LIN {X 0,Y 324.27,Z 263.767,A -85,B 0,C 180,E1 -15871.54,E2 -15871.54} C_VEL
LIN {X 0,Y 321.442,Z 259.609,A -85,B 0,C 180,E1 -15872.86,E2 -15872.86} C_VEL
LIN {X 0,Y 318.492,Z 255.533,A -85,B 0,C 180,E1 -15874.441,E2 -15874.441} C_VEL
LIN {X 0,Y 315.534,Z 252.043,A -85,B 0,C 180,E1 -15876.317,E2 -15876.317} C_VEL
LIN {X 0,Y 314.496,Z 250.773,A -85,B 0,C 180,E1 -15877.111,E2 -15877.111} C_VEL
LIN {X 0,Y 311.264,Z 247.746,A -85,B 0,C 180,E1 -15880.434,E2 -15880.434} C_VEL
LIN {X 0,Y 310.658,Z 246.885,A -85,B 0,C 180,E1 -15881.705,E2 -15881.705} C_VEL
LIN {X 0,Y 310.882,Z 247.509,A -85,B 0,C 180,E1 -15884.492,E2 -15884.492} C_VEL
LIN {X 0,Y 311.343,Z 249.074,A -85,B 0,C 180,E1 -15887.373,E2 -15887.373} C_VEL
LIN {X 0,Y 311.812,Z 250.468,A -85,B 0,C 180,E1 -15888.852,E2 -15888.852} C_VEL
LIN {X 0,Y 315.445,Z 256.63,A -85,B 0,C 180,E1 -15892.27,E2 -15892.27} C_VEL
LIN {X 0,Y 317.186,Z 259.203,A -85,B 0,C 180,E1 -15893.415,E2 -15893.415} C_VEL
LIN {X 0,Y 321.138,Z 266.17,A -85,B 0,C 180,E1 -15895.657,E2 -15895.657} C_VEL
LIN {X 0,Y 324.404,Z 272.439,A -85,B 0,C 180,E1 -15897.229,E2 -15897.229} C_VEL
LIN {X 0,Y 327.131,Z 278.303,A -85,B 0,C 180,E1 -15898.426,E2 -15898.426} C_VEL
LIN {X 0,Y 329.213,Z 283.156,A -85,B 0,C 180,E1 -15899.287,E2 -15899.287} C_VEL
LIN {X 0,Y 330.879,Z 295.045,A -85,B 0,C 180,E1 -15900.451,E2 -15900.451} C_VEL
LIN {X 0,Y 331.883,Z 305.844,A -85,B 0,C 180,E1 -15901.326,E2 -15901.326} C_VEL
LIN {X 0,Y 331.943,Z 308.748,A -85,B 0,C 180,E1 -15901.513,E2 -15901.513} C_VEL
LIN {X 0,Y 325.93,Z 368.1,A -85,B 0,C 180,E1 -15903.808,E2 -15903.808} C_VEL
LIN {X 0,Y 323.729,Z 382.809,A -85,B 0,C 180,E1 -15904.61,E2 -15904.61} C_VEL
LIN {X 0,Y 321.291,Z 396.25,A -85,B 0,C 180,E1 -15905.613,E2 -15905.613} C_VEL
LIN {X 0,Y 318.7,Z 408.35,A -85,B 0,C 180,E1 -15906.784,E2 -15906.784} C_VEL
LIN {X 0,Y 316.184,Z 419.438,A -85,B 0,C 180,E1 -15908.14,E2 -15908.14} C_VEL
LIN {X 0,Y 313.663,Z 429.65,A -85,B 0,C 180,E1 -15909.677,E2 -15909.677} C_VEL
LIN {X 0,Y 311.064,Z 439.677,A -85,B 0,C 180,E1 -15911.559,E2 -15911.559} C_VEL
LIN {X 0,Y 308.863,Z 447.905,A -85,B 0,C 180,E1 -15913.474,E2 -15913.474} C_VEL
LIN {X 0,Y 307.172,Z 454.592,A -85,B 0,C 180,E1 -15915.422,E2 -15915.422} C_VEL
LIN {X 0,Y 305.752,Z 460.004,A -85,B 0,C 180,E1 -15917.385,E2 -15917.385} C_VEL
LIN {X 0,Y 304.767,Z 464.279,A -85,B 0,C 180,E1 -15919.368,E2 -15919.368} C_VEL
LIN {X 0,Y 304.309,Z 466.526,A -85,B 0,C 180,E1 -15920.695,E2 -15920.695} C_VEL
LIN {X 0,Y 303.954,Z 468.349,A -85,B 0,C 180,E1 -15922.024,E2 -15922.024} C_VEL
LIN {X 0,Y 303.66,Z 470.501,A -85,B 0,C 180,E1 -15924.387,E2 -15924.387} C_VEL
LIN {X 0,Y 303.654,Z 471.167,A -85,B 0,C 180,E1 -15926.017,E2 -15926.017} C_VEL
LIN {X 0,Y 303.655,Z 471.261,A -85,B 0,C 180,E1 -15927.345,E2 -15927.345} C_VEL
LIN {X 0,Y 303.985,Z 470.229,A -85,B 0,C 180,E1 -15929.999,E2 -15929.999} C_VEL
LIN {X 0,Y 303.726,Z 470.328,A -85,B 0,C 180,E1 -15932.651,E2 -15932.651} C_VEL
LIN {X 0,Y 303.689,Z 469.744,A -85,B 0,C 180,E1 -15933.98,E2 -15933.98} C_VEL
LIN {X 0,Y 303.728,Z 468.388,A -85,B 0,C 180,E1 -15935.742,E2 -15935.742} C_VEL
LIN {X 0,Y 303.923,Z 465.595,A -85,B 0,C 180,E1 -15937.974,E2 -15937.974} C_VEL
LIN {X 0,Y 304.374,Z 462.049,A -85,B 0,C 180,E1 -15939.971,E2 -15939.971} C_VEL
LIN {X 0,Y 305.1,Z 457.403,A -85,B 0,C 180,E1 -15941.964,E2 -15941.964} C_VEL
LIN {X 0,Y 306.576,Z 450.407,A -85,B 0,C 180,E1 -15944.265,E2 -15944.265} C_VEL
LIN {X 0,Y 308.034,Z 442.766,A -85,B 0,C 180,E1 -15946.251,E2 -15946.251} C_VEL
LIN {X 0,Y 309.524,Z 435.145,A -85,B 0,C 180,E1 -15947.849,E2 -15947.849} C_VEL
LIN {X 0,Y 311.634,Z 424.665,A -85,B 0,C 180,E1 -15949.599,E2 -15949.599} C_VEL
LIN {X 0,Y 313.577,Z 414.013,A -85,B 0,C 180,E1 -15951.012,E2 -15951.012} C_VEL
LIN {X 0,Y 315.419,Z 401.913,A -85,B 0,C 180,E1 -15952.257,E2 -15952.257} C_VEL
LIN {X 0,Y 317.041,Z 390.09,A -85,B 0,C 180,E1 -15953.169,E2 -15953.169} C_VEL
LIN {X 0,Y 318.385,Z 378.012,A -85,B 0,C 180,E1 -15953.841,E2 -15953.841} C_VEL
LIN {X 0,Y 319.265,Z 364.396,A -85,B 0,C 180,E1 -15954.332,E2 -15954.332} C_VEL
LIN {X 0,Y 320.858,Z 303.853,A -85,B 0,C 180,E1 -15955.738,E2 -15955.738} C_VEL
LIN {X 0,Y 317.941,Z 282.581,A -85,B 0,C 180,E1 -15956.599,E2 -15956.599} C_VEL
LIN {X 0,Y 313.357,Z 256.247,A -85,B 0,C 180,E1 -15957.81,E2 -15957.81} C_VEL
LIN {X 0,Y 310.41,Z 248.436,A -85,B 0,C 180,E1 -15958.367,E2 -15958.367} C_VEL
LIN {X 0,Y 306.974,Z 238.832,A -85,B 0,C 180,E1 -15959.129,E2 -15959.129} C_VEL
LIN {X 0,Y 305.494,Z 231.423,A -85,B 0,C 180,E1 -15961.306,E2 -15961.306} C_VEL
LIN {X 0,Y 305.457,Z 231.411,A -85,B 0,C 180,E1 -15965.112,E2 -15965.112} C_VEL
LIN {X 0,Y 305.405,Z 231.432,A -85,B 0,C 180,E1 -15968.518,E2 -15968.518} C_VEL
LIN {X 0,Y 305.429,Z 231.43,A -85,B 0,C 180,E1 -15972.581,E2 -15972.581} C_VEL
LIN {X 0,Y 305.415,Z 231.439,A -85,B 0,C 180,E1 -15976.343,E2 -15976.343} C_VEL
LIN {X 0,Y 305.402,Z 231.436,A -85,B 0,C 180,E1 -15979.884,E2 -15979.884} C_VEL
LIN {X 0,Y 305.455,Z 231.413,A -85,B 0,C 180,E1 -15983.635,E2 -15983.635} C_VEL
LIN {X 0,Y 305.457,Z 231.429,A -85,B 0,C 180,E1 -15986.482,E2 -15986.482} C_VEL
LIN {X 0,Y 305.409,Z 231.42,A -85,B 0,C 180,E1 -15989.585,E2 -15989.585} C_VEL
LIN {X 0,Y 305.438,Z 231.423,A -85,B 0,C 180,E1 -15992.601,E2 -15992.601} C_VEL
LIN {X 0,Y 305.464,Z 231.423,A -85,B 0,C 180,E1 -15995.535,E2 -15995.535} C_VEL
LIN {X 0,Y 305.454,Z 231.402,A -85,B 0,C 180,E1 -15998.4,E2 -15998.4} C_VEL
LIN {X 0,Y 305.526,Z 231.425,A -85,B 0,C 180,E1 -16002.6,E2 -16002.6} C_VEL
LIN {X 0,Y 305.617,Z 231.385,A -85,B 0,C 180,E1 -16005.348,E2 -16005.348} C_VEL
LIN {X 0,Y 305.615,Z 231.414,A -85,B 0,C 180,E1 -16009.399,E2 -16009.399} C_VEL
LIN {X 0,Y 305.736,Z 231.392,A -85,B 0,C 180,E1 -16012.073,E2 -16012.073} C_VEL
LIN {X 0,Y 305.651,Z 231.378,A -85,B 0,C 180,E1 -16014.723,E2 -16014.723} C_VEL
LIN {X 0,Y 305.929,Z 231.374,A -85,B 0,C 180,E1 -16018.684,E2 -16018.684} C_VEL
LIN {X 0,Y 305.94,Z 231.353,A -85,B 0,C 180,E1 -16021.317,E2 -16021.317} C_VEL
LIN {X 0,Y 305.833,Z 231.384,A -85,B 0,C 180,E1 -16026.598,E2 -16026.598} C_VEL
LIN {X 0,Y 305.696,Z 231.382,A -85,B 0,C 180,E1 -16029.261,E2 -16029.261} C_VEL
LIN {X 0,Y 305.579,Z 231.414,A -85,B 0,C 180,E1 -16033.297,E2 -16033.297} C_VEL
LIN {X 0,Y 305.544,Z 231.409,A -85,B 0,C 180,E1 -16036.023,E2 -16036.023} C_VEL
LIN {X 0,Y 305.54,Z 231.417,A -85,B 0,C 180,E1 -16039.43,E2 -16039.43} C_VEL
LIN {X 0,Y 305.484,Z 231.417,A -85,B 0,C 180,E1 -16043.042,E2 -16043.042} C_VEL
LIN {X 0,Y 305.54,Z 231.425,A -85,B 0,C 180,E1 -16046.228,E2 -16046.228} C_VEL
LIN {X 0,Y 305.481,Z 231.419,A -85,B 0,C 180,E1 -16049.048,E2 -16049.048} C_VEL
LIN {X 0,Y 305.436,Z 231.44,A -85,B 0,C 180,E1 -16051.954,E2 -16051.954} C_VEL
LIN {X 0,Y 305.457,Z 231.43,A -85,B 0,C 180,E1 -16055.114,E2 -16055.114} C_VEL
LIN {X 0,Y 305.445,Z 231.43,A -85,B 0,C 180,E1 -16058.53,E2 -16058.53} C_VEL
LIN {X 0,Y 305.452,Z 231.432,A -85,B 0,C 180,E1 -16062.588,E2 -16062.588} C_VEL
LIN {X 0,Y 305.409,Z 231.439,A -85,B 0,C 180,E1 -16066.937,E2 -16066.937} C_VEL
LIN {X 0,Y 306.456,Z 234.33,A -85,B 0,C 180,E1 -16067.175,E2 -16067.175} C_VEL
LIN {X 0,Y 308.07,Z 236.957,A -85,B 0,C 180,E1 -16067.448,E2 -16067.448} C_VEL
LIN {X 0,Y 316.648,Z 252.215,A -85,B 0,C 180,E1 -16068.873,E2 -16068.873} C_VEL
LIN {X 0,Y 322.599,Z 264.535,A -85,B 0,C 180,E1 -16069.845,E2 -16069.845} C_VEL
LIN {X 0,Y 320.216,Z 341.058,A -85,B 0,C 180,E1 -16071.589,E2 -16071.589} C_VEL
LIN {X 0,Y 319.435,Z 354.384,A -85,B 0,C 180,E1 -16072.142,E2 -16072.142} C_VEL
LIN {X 0,Y 318.476,Z 365.661,A -85,B 0,C 180,E1 -16072.842,E2 -16072.842} C_VEL
LIN {X 0,Y 317.019,Z 377.635,A -85,B 0,C 180,E1 -16073.827,E2 -16073.827} C_VEL
LIN {X 0,Y 315.458,Z 388.546,A -85,B 0,C 180,E1 -16074.994,E2 -16074.994} C_VEL
LIN {X 0,Y 313.687,Z 398.497,A -85,B 0,C 180,E1 -16076.325,E2 -16076.325} C_VEL
LIN {X 0,Y 311.761,Z 408.517,A -85,B 0,C 180,E1 -16078.013,E2 -16078.013} C_VEL
LIN {X 0,Y 310.025,Z 416.996,A -85,B 0,C 180,E1 -16079.795,E2 -16079.795} C_VEL
LIN {X 0,Y 308.34,Z 424.504,A -85,B 0,C 180,E1 -16081.776,E2 -16081.776} C_VEL
LIN {X 0,Y 307.033,Z 430.143,A -85,B 0,C 180,E1 -16083.635,E2 -16083.635} C_VEL
LIN {X 0,Y 305.974,Z 434.812,A -85,B 0,C 180,E1 -16085.58,E2 -16085.58} C_VEL
LIN {X 0,Y 305.06,Z 438.66,A -85,B 0,C 180,E1 -16087.692,E2 -16087.692} C_VEL
LIN {X 0,Y 304.37,Z 441.306,A -85,B 0,C 180,E1 -16089.737,E2 -16089.737} C_VEL
LIN {X 0,Y 303.992,Z 442.756,A -85,B 0,C 180,E1 -16091.422,E2 -16091.422} C_VEL
LIN {X 0,Y 303.63,Z 443.679,A -85,B 0,C 180,E1 -16093.875,E2 -16093.875} C_VEL
LIN {X 0,Y 303.576,Z 443.218,A -85,B 0,C 180,E1 -16096.493,E2 -16096.493} C_VEL
LIN {X 0,Y 303.6,Z 442.239,A -85,B 0,C 180,E1 -16097.976,E2 -16097.976} C_VEL
LIN {X 0,Y 303.652,Z 440.927,A -85,B 0,C 180,E1 -16099.331,E2 -16099.331} C_VEL
LIN {X 0,Y 303.933,Z 438.132,A -85,B 0,C 180,E1 -16101.357,E2 -16101.357} C_VEL
LIN {X 0,Y 304.331,Z 434.302,A -85,B 0,C 180,E1 -16103.371,E2 -16103.371} C_VEL
LIN {X 0,Y 304.804,Z 429.35,A -85,B 0,C 180,E1 -16105.373,E2 -16105.373} C_VEL
LIN {X 0,Y 305.504,Z 423.101,A -85,B 0,C 180,E1 -16107.364,E2 -16107.364} C_VEL
LIN {X 0,Y 306.468,Z 415.263,A -85,B 0,C 180,E1 -16109.344,E2 -16109.344} C_VEL
LIN {X 0,Y 307.432,Z 407.282,A -85,B 0,C 180,E1 -16110.984,E2 -16110.984} C_VEL
LIN {X 0,Y 308.623,Z 397.563,A -85,B 0,C 180,E1 -16112.612,E2 -16112.612} C_VEL
LIN {X 0,Y 309.875,Z 386.849,A -85,B 0,C 180,E1 -16114.037,E2 -16114.037} C_VEL
LIN {X 0,Y 310.915,Z 375.975,A -85,B 0,C 180,E1 -16115.189,E2 -16115.189} C_VEL
LIN {X 0,Y 311.705,Z 364.413,A -85,B 0,C 180,E1 -16116.149,E2 -16116.149} C_VEL
LIN {X 0,Y 312.482,Z 351.83,A -85,B 0,C 180,E1 -16116.904,E2 -16116.904} C_VEL
LIN {X 0,Y 312.982,Z 338.785,A -85,B 0,C 180,E1 -16117.42,E2 -16117.42} C_VEL
LIN {X 0,Y 314.728,Z 259.21,A -85,B 0,C 180,E1 -16119.23,E2 -16119.23} C_VEL
LIN {X 0,Y 313.342,Z 251.333,A -85,B 0,C 180,E1 -16119.507,E2 -16119.507} C_VEL
LIN {X 0,Y 306.45,Z 233.925,A -85,B 0,C 180,E1 -16120.389,E2 -16120.389} C_VEL
LIN {X 0,Y 305.654,Z 231.414,A -85,B 0,C 180,E1 -16120.548,E2 -16120.548} C_VEL
LIN {X 0,Y 305.644,Z 231.411,A -85,B 0,C 180,E1 -16125.036,E2 -16125.036} C_VEL
LIN {X 0,Y 305.586,Z 231.419,A -85,B 0,C 180,E1 -16128.784,E2 -16128.784} C_VEL
LIN {X 0,Y 305.477,Z 231.43,A -85,B 0,C 180,E1 -16133.033,E2 -16133.033} C_VEL
LIN {X 0,Y 305.458,Z 231.436,A -85,B 0,C 180,E1 -16136.191,E2 -16136.191} C_VEL
LIN {X 0,Y 305.431,Z 231.437,A -85,B 0,C 180,E1 -16139.027,E2 -16139.027} C_VEL
LIN {X 0,Y 305.443,Z 231.439,A -85,B 0,C 180,E1 -16141.954,E2 -16141.954} C_VEL
LIN {X 0,Y 305.467,Z 231.432,A -85,B 0,C 180,E1 -16145.114,E2 -16145.114} C_VEL
LIN {X 0,Y 305.439,Z 231.436,A -85,B 0,C 180,E1 -16148.525,E2 -16148.525} C_VEL
LIN {X 0,Y 305.44,Z 231.432,A -85,B 0,C 180,E1 -16152.582,E2 -16152.582} C_VEL
LIN {X 0,Y 305.426,Z 231.437,A -85,B 0,C 180,E1 -16156.344,E2 -16156.344} C_VEL
LIN {X 0,Y 305.4,Z 231.439,A -85,B 0,C 180,E1 -16159.037,E2 -16159.037} C_VEL
LIN {X 0,Y 304.753,Z 231.522,A -85,B 0,C 180,E1 -16160.138,E2 -16160.138} C_VEL
LIN {X 0,Y 301.902,Z 231.875,A -85,B 0,C 180,E1 -16161.931,E2 -16161.931} C_VEL
LIN {X 0,Y 299.485,Z 232.178,A -85,B 0,C 180,E1 -16163.386,E2 -16163.386} C_VEL
LIN {X 0,Y 298.469,Z 232.303,A -85,B 0,C 180,E1 -16164.513,E2 -16164.513} C_VEL
LIN {X 0,Y 298.398,Z 232.309,A -85,B 0,C 180,E1 -16164.894,E2 -16164.894} C_VEL
LIN {X 0,Y 298.377,Z 232.317,A -85,B 0,C 180,E1 -16168.789,E2 -16168.789} C_VEL
LIN {X 0,Y 298.41,Z 232.302,A -85,B 0,C 180,E1 -16171.898,E2 -16171.898} C_VEL
LIN {X 0,Y 298.471,Z 232.351,A -85,B 0,C 180,E1 -16175.457,E2 -16175.457} C_VEL
LIN {X 0,Y 298.728,Z 233.608,A -85,B 0,C 180,E1 -16175.791,E2 -16175.791} C_VEL
LIN {X 0,Y 304.574,Z 256.081,A -85,B 0,C 180,E1 -16176.845,E2 -16176.845} C_VEL
LIN {X 0,Y 305.328,Z 261.998,A -85,B 0,C 180,E1 -16177.086,E2 -16177.086} C_VEL
LIN {X 0,Y 302.456,Z 342.479,A -85,B 0,C 180,E1 -16179.911,E2 -16179.911} C_VEL
LIN {X 0,Y 301.986,Z 355.703,A -85,B 0,C 180,E1 -16180.632,E2 -16180.632} C_VEL
LIN {X 0,Y 301.269,Z 369.111,A -85,B 0,C 180,E1 -16181.643,E2 -16181.643} C_VEL
LIN {X 0,Y 300.468,Z 381.148,A -85,B 0,C 180,E1 -16182.824,E2 -16182.824} C_VEL
LIN {X 0,Y 299.696,Z 391.71,A -85,B 0,C 180,E1 -16184.116,E2 -16184.116} C_VEL
LIN {X 0,Y 298.948,Z 402.266,A -85,B 0,C 180,E1 -16185.709,E2 -16185.709} C_VEL
LIN {X 0,Y 298.245,Z 411.532,A -85,B 0,C 180,E1 -16187.41,E2 -16187.41} C_VEL
LIN {X 0,Y 297.714,Z 419.213,A -85,B 0,C 180,E1 -16189.114,E2 -16189.114} C_VEL
LIN {X 0,Y 297.237,Z 426.724,A -85,B 0,C 180,E1 -16191.159,E2 -16191.159} C_VEL
LIN {X 0,Y 296.932,Z 432.717,A -85,B 0,C 180,E1 -16193.203,E2 -16193.203} C_VEL
LIN {X 0,Y 296.744,Z 437.411,A -85,B 0,C 180,E1 -16195.245,E2 -16195.245} C_VEL
LIN {X 0,Y 296.681,Z 440.952,A -85,B 0,C 180,E1 -16197.284,E2 -16197.284} C_VEL
LIN {X 0,Y 296.631,Z 442.74,A -85,B 0,C 180,E1 -16198.642,E2 -16198.642} C_VEL
LIN {X 0,Y 296.695,Z 444.045,A -85,B 0,C 180,E1 -16200,E2 -16200} C_VEL
LIN {X 0,Y 296.858,Z 444.911,A -85,B 0,C 180,E1 -16201.356,E2 -16201.356} C_VEL
LIN {X 0,Y 297.102,Z 445.37,A -85,B 0,C 180,E1 -16202.711,E2 -16202.711} C_VEL
LIN {X 0,Y 297.47,Z 445.402,A -85,B 0,C 180,E1 -16204.064,E2 -16204.064} C_VEL
LIN {X 0,Y 297.933,Z 444.971,A -85,B 0,C 180,E1 -16205.414,E2 -16205.414} C_VEL
LIN {X 0,Y 298.231,Z 444.155,A -85,B 0,C 180,E1 -16206.767,E2 -16206.767} C_VEL
LIN {X 0,Y 298.552,Z 442.95,A -85,B 0,C 180,E1 -16208.119,E2 -16208.119} C_VEL
LIN {X 0,Y 300.197,Z 439.612,A -85,B 0,C 180,E1 -16210.487,E2 -16210.487} C_VEL
LIN {X 0,Y 301.927,Z 434.969,A -85,B 0,C 180,E1 -16212.775,E2 -16212.775} C_VEL
LIN {X 0,Y 304.13,Z 428.717,A -85,B 0,C 180,E1 -16215.068,E2 -16215.068} C_VEL
LIN {X 0,Y 306.32,Z 421.893,A -85,B 0,C 180,E1 -16217.009,E2 -16217.009} C_VEL
LIN {X 0,Y 308.873,Z 413.464,A -85,B 0,C 180,E1 -16218.919,E2 -16218.919} C_VEL
LIN {X 0,Y 311.286,Z 404.929,A -85,B 0,C 180,E1 -16220.484,E2 -16220.484} C_VEL
LIN {X 0,Y 313.958,Z 394.59,A -85,B 0,C 180,E1 -16222.021,E2 -16222.021} C_VEL
LIN {X 0,Y 316.768,Z 381.851,A -85,B 0,C 180,E1 -16223.538,E2 -16223.538} C_VEL
LIN {X 0,Y 319.27,Z 368.719,A -85,B 0,C 180,E1 -16224.723,E2 -16224.723} C_VEL
LIN {X 0,Y 321.125,Z 356.231,A -85,B 0,C 180,E1 -16225.61,E2 -16225.61} C_VEL
LIN {X 0,Y 322.948,Z 340.967,A -85,B 0,C 180,E1 -16226.364,E2 -16226.364} C_VEL
LIN {X 0,Y 329.392,Z 284.527,A -85,B 0,C 180,E1 -16228.59,E2 -16228.59} C_VEL
LIN {X 0,Y 325.775,Z 277.054,A -85,B 0,C 180,E1 -16230.035,E2 -16230.035} C_VEL
LIN {X 0,Y 321.791,Z 270.367,A -85,B 0,C 180,E1 -16231.752,E2 -16231.752} C_VEL
LIN {X 0,Y 318.626,Z 265.727,A -85,B 0,C 180,E1 -16233.288,E2 -16233.288} C_VEL
LIN {X 0,Y 315.758,Z 261.708,A -85,B 0,C 180,E1 -16234.924,E2 -16234.924} C_VEL
LIN {X 0,Y 313.045,Z 258.146,A -85,B 0,C 180,E1 -16236.827,E2 -16236.827} C_VEL
LIN {X 0,Y 311.199,Z 256.452,A -85,B 0,C 180,E1 -16238.376,E2 -16238.376} C_VEL
LIN {X 0,Y 309.035,Z 253.983,A -85,B 0,C 180,E1 -16241.366,E2 -16241.366} C_VEL
LIN {X 0,Y 308.261,Z 254.006,A -85,B 0,C 180,E1 -16244.08,E2 -16244.08} C_VEL
LIN {X 0,Y 308.771,Z 255.362,A -85,B 0,C 180,E1 -16246.749,E2 -16246.749} C_VEL
LIN {X 0,Y 309.859,Z 257.192,A -85,B 0,C 180,E1 -16248.618,E2 -16248.618} C_VEL
LIN {X 0,Y 313.257,Z 263.264,A -85,B 0,C 180,E1 -16252.027,E2 -16252.027} C_VEL
LIN {X 0,Y 314.664,Z 265.534,A -85,B 0,C 180,E1 -16253.024,E2 -16253.024} C_VEL
LIN {X 0,Y 318.17,Z 272.075,A -85,B 0,C 180,E1 -16255.176,E2 -16255.176} C_VEL
LIN {X 0,Y 321.172,Z 278.16,A -85,B 0,C 180,E1 -16256.732,E2 -16256.732} C_VEL
LIN {X 0,Y 323.667,Z 283.829,A -85,B 0,C 180,E1 -16257.919,E2 -16257.919} C_VEL
LIN {X 0,Y 325.18,Z 287.739,A -85,B 0,C 180,E1 -16258.614,E2 -16258.614} C_VEL
LIN {X 0,Y 326.58,Z 299.644,A -85,B 0,C 180,E1 -16259.794,E2 -16259.794} C_VEL
LIN {X 0,Y 327.257,Z 309.221,A -85,B 0,C 180,E1 -16260.574,E2 -16260.574} C_VEL
LIN {X 0,Y 320.93,Z 367.302,A -85,B 0,C 180,E1 -16262.884,E2 -16262.884} C_VEL
LIN {X 0,Y 318.79,Z 381.297,A -85,B 0,C 180,E1 -16263.66,E2 -16263.66} C_VEL
LIN {X 0,Y 316.461,Z 393.138,A -85,B 0,C 180,E1 -16264.513,E2 -16264.513} C_VEL
LIN {X 0,Y 313.705,Z 405.712,A -85,B 0,C 180,E1 -16265.689,E2 -16265.689} C_VEL
LIN {X 0,Y 310.879,Z 417.125,A -85,B 0,C 180,E1 -16267.046,E2 -16267.046} C_VEL
LIN {X 0,Y 308.187,Z 427.579,A -85,B 0,C 180,E1 -16268.599,E2 -16268.599} C_VEL
LIN {X 0,Y 305.749,Z 436.315,A -85,B 0,C 180,E1 -16270.18,E2 -16270.18} C_VEL
LIN {X 0,Y 303.163,Z 445.032,A -85,B 0,C 180,E1 -16272.113,E2 -16272.113} C_VEL
LIN {X 0,Y 301.249,Z 452.123,A -85,B 0,C 180,E1 -16274.089,E2 -16274.089} C_VEL
LIN {X 0,Y 299.216,Z 458.804,A -85,B 0,C 180,E1 -16276.414,E2 -16276.414} C_VEL
LIN {X 0,Y 298.098,Z 463.24,A -85,B 0,C 180,E1 -16278.438,E2 -16278.438} C_VEL
LIN {X 0,Y 297.281,Z 466.614,A -85,B 0,C 180,E1 -16280.473,E2 -16280.473} C_VEL
LIN {X 0,Y 296.895,Z 468.311,A -85,B 0,C 180,E1 -16281.833,E2 -16281.833} C_VEL
LIN {X 0,Y 296.588,Z 470.328,A -85,B 0,C 180,E1 -16284.406,E2 -16284.406} C_VEL
LIN {X 0,Y 296.568,Z 470.839,A -85,B 0,C 180,E1 -16285.922,E2 -16285.922} C_VEL
LIN {X 0,Y 296.578,Z 470.815,A -85,B 0,C 180,E1 -16287.282,E2 -16287.282} C_VEL
LIN {X 0,Y 296.889,Z 469.87,A -85,B 0,C 180,E1 -16289.999,E2 -16289.999} C_VEL
LIN {X 0,Y 296.644,Z 470.033,A -85,B 0,C 180,E1 -16292.714,E2 -16292.714} C_VEL
LIN {X 0,Y 296.603,Z 469.487,A -85,B 0,C 180,E1 -16294.075,E2 -16294.075} C_VEL
LIN {X 0,Y 296.622,Z 468.346,A -85,B 0,C 180,E1 -16295.659,E2 -16295.659} C_VEL
LIN {X 0,Y 296.862,Z 465.434,A -85,B 0,C 180,E1 -16298.165,E2 -16298.165} C_VEL
LIN {X 0,Y 297.361,Z 461.943,A -85,B 0,C 180,E1 -16300.209,E2 -16300.209} C_VEL
LIN {X 0,Y 298.121,Z 457.363,A -85,B 0,C 180,E1 -16302.248,E2 -16302.248} C_VEL
LIN {X 0,Y 299.691,Z 450.436,A -85,B 0,C 180,E1 -16304.6,E2 -16304.6} C_VEL
LIN {X 0,Y 301.158,Z 443.106,A -85,B 0,C 180,E1 -16306.573,E2 -16306.573} C_VEL
LIN {X 0,Y 302.781,Z 435.35,A -85,B 0,C 180,E1 -16308.26,E2 -16308.26} C_VEL
LIN {X 0,Y 304.754,Z 426.07,A -85,B 0,C 180,E1 -16309.885,E2 -16309.885} C_VEL
LIN {X 0,Y 306.792,Z 415.77,A -85,B 0,C 180,E1 -16311.324,E2 -16311.324} C_VEL
LIN {X 0,Y 308.654,Z 404.364,A -85,B 0,C 180,E1 -16312.595,E2 -16312.595} C_VEL
LIN {X 0,Y 310.435,Z 392.286,A -85,B 0,C 180,E1 -16313.603,E2 -16313.603} C_VEL
LIN {X 0,Y 312.032,Z 378.901,A -85,B 0,C 180,E1 -16314.402,E2 -16314.402} C_VEL
LIN {X 0,Y 312.967,Z 366.327,A -85,B 0,C 180,E1 -16314.899,E2 -16314.899} C_VEL
LIN {X 0,Y 314.722,Z 304.889,A -85,B 0,C 180,E1 -16316.36,E2 -16316.36} C_VEL
LIN {X 0,Y 312.132,Z 285.348,A -85,B 0,C 180,E1 -16317.168,E2 -16317.168} C_VEL
LIN {X 0,Y 307.592,Z 258.654,A -85,B 0,C 180,E1 -16318.424,E2 -16318.424} C_VEL
LIN {X 0,Y 301.295,Z 242.01,A -85,B 0,C 180,E1 -16319.725,E2 -16319.725} C_VEL
LIN {X 0,Y 299.357,Z 236.961,A -85,B 0,C 180,E1 -16320.186,E2 -16320.186} C_VEL
LIN {X 0,Y 299.192,Z 236.151,A -85,B 0,C 180,E1 -16320.29,E2 -16320.29} C_VEL
LIN {X 0,Y 298.455,Z 232.294,A -85,B 0,C 180,E1 -16321.49,E2 -16321.49} C_VEL
LIN {X 0,Y 298.423,Z 232.277,A -85,B 0,C 180,E1 -16324.486,E2 -16324.486} C_VEL
LIN {X 0,Y 298.386,Z 232.313,A -85,B 0,C 180,E1 -16327.76,E2 -16327.76} C_VEL
LIN {X 0,Y 298.342,Z 232.324,A -85,B 0,C 180,E1 -16331.266,E2 -16331.266} C_VEL
LIN {X 0,Y 298.348,Z 232.319,A -85,B 0,C 180,E1 -16335.034,E2 -16335.034} C_VEL
LIN {X 0,Y 298.34,Z 232.305,A -85,B 0,C 180,E1 -16338.92,E2 -16338.92} C_VEL
LIN {X 0,Y 298.391,Z 232.31,A -85,B 0,C 180,E1 -16342.238,E2 -16342.238} C_VEL
LIN {X 0,Y 298.4,Z 232.299,A -85,B 0,C 180,E1 -16345.58,E2 -16345.58} C_VEL
LIN {X 0,Y 298.364,Z 232.305,A -85,B 0,C 180,E1 -16348.788,E2 -16348.788} C_VEL
LIN {X 0,Y 298.39,Z 232.293,A -85,B 0,C 180,E1 -16351.897,E2 -16351.897} C_VEL
LIN {X 0,Y 298.429,Z 232.305,A -85,B 0,C 180,E1 -16354.919,E2 -16354.919} C_VEL
LIN {X 0,Y 298.391,Z 232.28,A -85,B 0,C 180,E1 -16357.862,E2 -16357.862} C_VEL
LIN {X 0,Y 298.455,Z 232.299,A -85,B 0,C 180,E1 -16360.751,E2 -16360.751} C_VEL
LIN {X 0,Y 298.577,Z 232.265,A -85,B 0,C 180,E1 -16364.994,E2 -16364.994} C_VEL
LIN {X 0,Y 298.574,Z 232.291,A -85,B 0,C 180,E1 -16369.146,E2 -16369.146} C_VEL
LIN {X 0,Y 298.688,Z 232.273,A -85,B 0,C 180,E1 -16371.884,E2 -16371.884} C_VEL
LIN {X 0,Y 298.621,Z 232.253,A -85,B 0,C 180,E1 -16374.598,E2 -16374.598} C_VEL
LIN {X 0,Y 298.897,Z 232.25,A -85,B 0,C 180,E1 -16378.653,E2 -16378.653} C_VEL
LIN {X 0,Y 298.906,Z 232.228,A -85,B 0,C 180,E1 -16381.348,E2 -16381.348} C_VEL
LIN {X 0,Y 298.778,Z 232.262,A -85,B 0,C 180,E1 -16386.755,E2 -16386.755} C_VEL
LIN {X 0,Y 298.627,Z 232.259,A -85,B 0,C 180,E1 -16389.483,E2 -16389.483} C_VEL
LIN {X 0,Y 298.538,Z 232.293,A -85,B 0,C 180,E1 -16393.616,E2 -16393.616} C_VEL
LIN {X 0,Y 298.479,Z 232.285,A -85,B 0,C 180,E1 -16396.413,E2 -16396.413} C_VEL
LIN {X 0,Y 298.481,Z 232.298,A -85,B 0,C 180,E1 -16399.643,E2 -16399.643} C_VEL
LIN {X 0,Y 298.451,Z 232.289,A -85,B 0,C 180,E1 -16403.599,E2 -16403.599} C_VEL
LIN {X 0,Y 298.483,Z 232.304,A -85,B 0,C 180,E1 -16406.576,E2 -16406.576} C_VEL
LIN {X 0,Y 298.41,Z 232.299,A -85,B 0,C 180,E1 -16409.643,E2 -16409.643} C_VEL
LIN {X 0,Y 298.389,Z 232.314,A -85,B 0,C 180,E1 -16412.802,E2 -16412.802} C_VEL
LIN {X 0,Y 298.442,Z 232.314,A -85,B 0,C 180,E1 -16416.809,E2 -16416.809} C_VEL
LIN {X 0,Y 298.382,Z 232.315,A -85,B 0,C 180,E1 -16421.089,E2 -16421.089} C_VEL
LIN {X 0,Y 298.394,Z 232.316,A -85,B 0,C 180,E1 -16423.105,E2 -16423.105} C_VEL
LIN {X 0,Y 298.36,Z 232.321,A -85,B 0,C 180,E1 -16426.047,E2 -16426.047} C_VEL
LIN {X 0,Y 299.336,Z 235.105,A -85,B 0,C 180,E1 -16426.278,E2 -16426.278} C_VEL
LIN {X 0,Y 301.106,Z 237.894,A -85,B 0,C 180,E1 -16426.593,E2 -16426.593} C_VEL
LIN {X 0,Y 310.001,Z 253.515,A -85,B 0,C 180,E1 -16428.137,E2 -16428.137} C_VEL
LIN {X 0,Y 316.428,Z 266.345,A -85,B 0,C 180,E1 -16429.222,E2 -16429.222} C_VEL
LIN {X 0,Y 314.031,Z 341.028,A -85,B 0,C 180,E1 -16430.956,E2 -16430.956} C_VEL
LIN {X 0,Y 313.272,Z 353.948,A -85,B 0,C 180,E1 -16431.49,E2 -16431.49} C_VEL
LIN {X 0,Y 312.243,Z 365.654,A -85,B 0,C 180,E1 -16432.216,E2 -16432.216} C_VEL
LIN {X 0,Y 310.778,Z 377.333,A -85,B 0,C 180,E1 -16433.184,E2 -16433.184} C_VEL
LIN {X 0,Y 309.151,Z 388.375,A -85,B 0,C 180,E1 -16434.373,E2 -16434.373} C_VEL
LIN {X 0,Y 307.297,Z 398.436,A -85,B 0,C 180,E1 -16435.726,E2 -16435.726} C_VEL
LIN {X 0,Y 305.422,Z 407.608,A -85,B 0,C 180,E1 -16437.267,E2 -16437.267} C_VEL
LIN {X 0,Y 303.614,Z 416.138,A -85,B 0,C 180,E1 -16439.048,E2 -16439.048} C_VEL
LIN {X 0,Y 301.772,Z 424.05,A -85,B 0,C 180,E1 -16441.104,E2 -16441.104} C_VEL
LIN {X 0,Y 300.283,Z 430.177,A -85,B 0,C 180,E1 -16443.132,E2 -16443.132} C_VEL
LIN {X 0,Y 299.204,Z 434.646,A -85,B 0,C 180,E1 -16444.99,E2 -16444.99} C_VEL
LIN {X 0,Y 298.395,Z 437.922,A -85,B 0,C 180,E1 -16446.717,E2 -16446.717} C_VEL
LIN {X 0,Y 297.424,Z 441.378,A -85,B 0,C 180,E1 -16449.242,E2 -16449.242} C_VEL
LIN {X 0,Y 296.943,Z 443.077,A -85,B 0,C 180,E1 -16451.213,E2 -16451.213} C_VEL
LIN {X 0,Y 296.578,Z 443.973,A -85,B 0,C 180,E1 -16453.481,E2 -16453.481} C_VEL
LIN {X 0,Y 296.465,Z 443.974,A -85,B 0,C 180,E1 -16454.886,E2 -16454.886} C_VEL
LIN {X 0,Y 296.478,Z 443.54,A -85,B 0,C 180,E1 -16456.389,E2 -16456.389} C_VEL
LIN {X 0,Y 296.493,Z 442.75,A -85,B 0,C 180,E1 -16457.684,E2 -16457.684} C_VEL
LIN {X 0,Y 296.537,Z 441.492,A -85,B 0,C 180,E1 -16459.072,E2 -16459.072} C_VEL
LIN {X 0,Y 296.799,Z 438.81,A -85,B 0,C 180,E1 -16461.148,E2 -16461.148} C_VEL
LIN {X 0,Y 297.213,Z 434.928,A -85,B 0,C 180,E1 -16463.294,E2 -16463.294} C_VEL
LIN {X 0,Y 297.672,Z 430.271,A -85,B 0,C 180,E1 -16465.262,E2 -16465.262} C_VEL
LIN {X 0,Y 298.382,Z 424.179,A -85,B 0,C 180,E1 -16467.301,E2 -16467.301} C_VEL
LIN {X 0,Y 299.348,Z 416.56,A -85,B 0,C 180,E1 -16469.329,E2 -16469.329} C_VEL
LIN {X 0,Y 300.543,Z 407.023,A -85,B 0,C 180,E1 -16471.341,E2 -16471.341} C_VEL
LIN {X 0,Y 301.81,Z 397.14,A -85,B 0,C 180,E1 -16473.005,E2 -16473.005} C_VEL
LIN {X 0,Y 303.157,Z 385.626,A -85,B 0,C 180,E1 -16474.535,E2 -16474.535} C_VEL
LIN {X 0,Y 304.165,Z 375.162,A -85,B 0,C 180,E1 -16475.637,E2 -16475.637} C_VEL
LIN {X 0,Y 305.006,Z 363.172,A -85,B 0,C 180,E1 -16476.617,E2 -16476.617} C_VEL
LIN {X 0,Y 305.755,Z 349.938,A -85,B 0,C 180,E1 -16477.389,E2 -16477.389} C_VEL
LIN {X 0,Y 306.284,Z 336.766,A -85,B 0,C 180,E1 -16477.873,E2 -16477.873} C_VEL
LIN {X 0,Y 307.978,Z 259.724,A -85,B 0,C 180,E1 -16479.652,E2 -16479.652} C_VEL
LIN {X 0,Y 306.668,Z 252.882,A -85,B 0,C 180,E1 -16479.906,E2 -16479.906} C_VEL
LIN {X 0,Y 298.672,Z 232.84,A -85,B 0,C 180,E1 -16480.961,E2 -16480.961} C_VEL
LIN {X 0,Y 298.574,Z 232.294,A -85,B 0,C 180,E1 -16481.027,E2 -16481.027} C_VEL
LIN {X 0,Y 298.612,Z 232.287,A -85,B 0,C 180,E1 -16485.21,E2 -16485.21} C_VEL
LIN {X 0,Y 298.531,Z 232.297,A -85,B 0,C 180,E1 -16489.245,E2 -16489.245} C_VEL
LIN {X 0,Y 298.415,Z 232.311,A -85,B 0,C 180,E1 -16493.603,E2 -16493.603} C_VEL
LIN {X 0,Y 298.407,Z 232.312,A -85,B 0,C 180,E1 -16496.584,E2 -16496.584} C_VEL
LIN {X 0,Y 298.364,Z 232.32,A -85,B 0,C 180,E1 -16499.649,E2 -16499.649} C_VEL
LIN {X 0,Y 298.399,Z 232.313,A -85,B 0,C 180,E1 -16502.801,E2 -16502.801} C_VEL
LIN {X 0,Y 298.432,Z 232.306,A -85,B 0,C 180,E1 -16506.803,E2 -16506.803} C_VEL
LIN {X 0,Y 298.38,Z 232.319,A -85,B 0,C 180,E1 -16509.493,E2 -16509.493} C_VEL
LIN {X 0,Y 298.375,Z 232.314,A -85,B 0,C 180,E1 -16513.098,E2 -16513.098} C_VEL
LIN {X 0,Y 298.376,Z 232.317,A -85,B 0,C 180,E1 -16516.915,E2 -16516.915} C_VEL
LIN {X 0,Y 298.36,Z 232.316,A -85,B 0,C 180,E1 -16521.019,E2 -16521.019} C_VEL
LIN {X 0,Y 298.41,Z 232.309,A -85,B 0,C 180,E1 -16523.928,E2 -16523.928} C_VEL
LIN {X 0,Y 298.398,Z 232.309,A -85,B 0,C 180,E1 -16524.894,E2 -16524.894} C_VEL
LIN {X 0,Y 297.758,Z 232.393,A -85,B 0,C 180,E1 -16526.02,E2 -16526.02} C_VEL
LIN {X 0,Y 294.899,Z 232.749,A -85,B 0,C 180,E1 -16527.852,E2 -16527.852} C_VEL
LIN {X 0,Y 292.457,Z 233.05,A -85,B 0,C 180,E1 -16529.339,E2 -16529.339} C_VEL
LIN {X 0,Y 291.409,Z 233.18,A -85,B 0,C 180,E1 -16530.491,E2 -16530.491} C_VEL
LIN {X 0,Y 291.325,Z 233.186,A -85,B 0,C 180,E1 -16530.882,E2 -16530.882} C_VEL
LIN {X 0,Y 291.443,Z 233.299,A -85,B 0,C 180,E1 -16535.371,E2 -16535.371} C_VEL
LIN {X 0,Y 291.494,Z 233.639,A -85,B 0,C 180,E1 -16535.486,E2 -16535.486} C_VEL
LIN {X 0,Y 297.767,Z 257.83,A -85,B 0,C 180,E1 -16536.648,E2 -16536.648} C_VEL
LIN {X 0,Y 298.399,Z 261.628,A -85,B 0,C 180,E1 -16536.813,E2 -16536.813} C_VEL
LIN {X 0,Y 295.424,Z 342.104,A -85,B 0,C 180,E1 -16539.73,E2 -16539.73} C_VEL
LIN {X 0,Y 294.93,Z 356.112,A -85,B 0,C 180,E1 -16540.511,E2 -16540.511} C_VEL
LIN {X 0,Y 294.194,Z 369.44,A -85,B 0,C 180,E1 -16541.546,E2 -16541.546} C_VEL
LIN {X 0,Y 293.388,Z 381.449,A -85,B 0,C 180,E1 -16542.756,E2 -16542.756} C_VEL
LIN {X 0,Y 292.557,Z 392.188,A -85,B 0,C 180,E1 -16544.101,E2 -16544.101} C_VEL
LIN {X 0,Y 291.834,Z 402.592,A -85,B 0,C 180,E1 -16545.709,E2 -16545.709} C_VEL
LIN {X 0,Y 291.11,Z 411.847,A -85,B 0,C 180,E1 -16547.45,E2 -16547.45} C_VEL
LIN {X 0,Y 290.6,Z 419.532,A -85,B 0,C 180,E1 -16549.197,E2 -16549.197} C_VEL
LIN {X 0,Y 290.121,Z 427.048,A -85,B 0,C 180,E1 -16551.291,E2 -16551.291} C_VEL
LIN {X 0,Y 289.746,Z 433.942,A -85,B 0,C 180,E1 -16553.734,E2 -16553.734} C_VEL
LIN {X 0,Y 289.663,Z 438.454,A -85,B 0,C 180,E1 -16555.826,E2 -16555.826} C_VEL
LIN {X 0,Y 289.609,Z 440.803,A -85,B 0,C 180,E1 -16557.218,E2 -16557.218} C_VEL
LIN {X 0,Y 289.548,Z 442.684,A -85,B 0,C 180,E1 -16558.609,E2 -16558.609} C_VEL
LIN {X 0,Y 289.604,Z 444.139,A -85,B 0,C 180,E1 -16560,E2 -16560} C_VEL
LIN {X 0,Y 289.767,Z 445.138,A -85,B 0,C 180,E1 -16561.389,E2 -16561.389} C_VEL
LIN {X 0,Y 290.018,Z 445.69,A -85,B 0,C 180,E1 -16562.778,E2 -16562.778} C_VEL
LIN {X 0,Y 290.402,Z 445.833,A -85,B 0,C 180,E1 -16564.163,E2 -16564.163} C_VEL
LIN {X 0,Y 290.881,Z 445.567,A -85,B 0,C 180,E1 -16565.546,E2 -16565.546} C_VEL
LIN {X 0,Y 291.203,Z 444.871,A -85,B 0,C 180,E1 -16566.931,E2 -16566.931} C_VEL
LIN {X 0,Y 291.581,Z 443.764,A -85,B 0,C 180,E1 -16568.315,E2 -16568.315} C_VEL
LIN {X 0,Y 293.356,Z 440.581,A -85,B 0,C 180,E1 -16570.806,E2 -16570.806} C_VEL
LIN {X 0,Y 295.154,Z 436.334,A -85,B 0,C 180,E1 -16573.074,E2 -16573.074} C_VEL
LIN {X 0,Y 297.094,Z 431.32,A -85,B 0,C 180,E1 -16575.083,E2 -16575.083} C_VEL
LIN {X 0,Y 299.769,Z 423.869,A -85,B 0,C 180,E1 -16577.393,E2 -16577.393} C_VEL
LIN {X 0,Y 302.48,Z 415.86,A -85,B 0,C 180,E1 -16579.335,E2 -16579.335} C_VEL
LIN {X 0,Y 305.512,Z 405.93,A -85,B 0,C 180,E1 -16581.242,E2 -16581.242} C_VEL
LIN {X 0,Y 308.366,Z 395.796,A -85,B 0,C 180,E1 -16582.796,E2 -16582.796} C_VEL
LIN {X 0,Y 311.338,Z 383.332,A -85,B 0,C 180,E1 -16584.328,E2 -16584.328} C_VEL
LIN {X 0,Y 314.001,Z 370.625,A -85,B 0,C 180,E1 -16585.522,E2 -16585.522} C_VEL
LIN {X 0,Y 316.164,Z 357.575,A -85,B 0,C 180,E1 -16586.485,E2 -16586.485} C_VEL
LIN {X 0,Y 318.178,Z 342.168,A -85,B 0,C 180,E1 -16587.279,E2 -16587.279} C_VEL
LIN {X 0,Y 324.886,Z 287.875,A -85,B 0,C 180,E1 -16589.457,E2 -16589.457} C_VEL
LIN {X 0,Y 321.204,Z 280.481,A -85,B 0,C 180,E1 -16591.056,E2 -16591.056} C_VEL
LIN {X 0,Y 317.994,Z 275.189,A -85,B 0,C 180,E1 -16592.581,E2 -16592.581} C_VEL
LIN {X 0,Y 315.92,Z 271.898,A -85,B 0,C 180,E1 -16593.691,E2 -16593.691} C_VEL
LIN {X 0,Y 313.409,Z 268.199,A -85,B 0,C 180,E1 -16595.224,E2 -16595.224} C_VEL
LIN {X 0,Y 310.841,Z 264.719,A -85,B 0,C 180,E1 -16597.129,E2 -16597.129} C_VEL
LIN {X 0,Y 307.917,Z 261.824,A -85,B 0,C 180,E1 -16600.15,E2 -16600.15} C_VEL
LIN {X 0,Y 307.185,Z 260.832,A -85,B 0,C 180,E1 -16601.566,E2 -16601.566} C_VEL
LIN {X 0,Y 306.519,Z 260.973,A -85,B 0,C 180,E1 -16604.396,E2 -16604.396} C_VEL
LIN {X 0,Y 307.153,Z 262.51,A -85,B 0,C 180,E1 -16607.071,E2 -16607.071} C_VEL
LIN {X 0,Y 307.971,Z 264.089,A -85,B 0,C 180,E1 -16608.498,E2 -16608.498} C_VEL
LIN {X 0,Y 311.216,Z 270.144,A -85,B 0,C 180,E1 -16611.905,E2 -16611.905} C_VEL
LIN {X 0,Y 312.178,Z 271.879,A -85,B 0,C 180,E1 -16612.643,E2 -16612.643} C_VEL
LIN {X 0,Y 315.263,Z 277.988,A -85,B 0,C 180,E1 -16614.687,E2 -16614.687} C_VEL
LIN {X 0,Y 317.837,Z 283.501,A -85,B 0,C 180,E1 -16616.139,E2 -16616.139} C_VEL
LIN {X 0,Y 320.384,Z 289.625,A -85,B 0,C 180,E1 -16617.454,E2 -16617.454} C_VEL
LIN {X 0,Y 321.277,Z 292.365,A -85,B 0,C 180,E1 -16617.924,E2 -16617.924} C_VEL
LIN {X 0,Y 322.371,Z 304.339,A -85,B 0,C 180,E1 -16619.114,E2 -16619.114} C_VEL
LIN {X 0,Y 322.659,Z 311.335,A -85,B 0,C 180,E1 -16619.673,E2 -16619.673} C_VEL
LIN {X 0,Y 315.991,Z 367.704,A -85,B 0,C 180,E1 -16621.974,E2 -16621.974} C_VEL
LIN {X 0,Y 313.73,Z 381.285,A -85,B 0,C 180,E1 -16622.751,E2 -16622.751} C_VEL
LIN {X 0,Y 311.454,Z 392.071,A -85,B 0,C 180,E1 -16623.533,E2 -16623.533} C_VEL
LIN {X 0,Y 308.527,Z 404.642,A -85,B 0,C 180,E1 -16624.714,E2 -16624.714} C_VEL
LIN {X 0,Y 305.522,Z 416.11,A -85,B 0,C 180,E1 -16626.08,E2 -16626.08} C_VEL
LIN {X 0,Y 302.314,Z 427.56,A -85,B 0,C 180,E1 -16627.803,E2 -16627.803} C_VEL
LIN {X 0,Y 299.207,Z 437.711,A -85,B 0,C 180,E1 -16629.728,E2 -16629.728} C_VEL
LIN {X 0,Y 296.537,Z 446.004,A -85,B 0,C 180,E1 -16631.678,E2 -16631.678} C_VEL
LIN {X 0,Y 294.472,Z 452.902,A -85,B 0,C 180,E1 -16633.713,E2 -16633.713} C_VEL
LIN {X 0,Y 292.339,Z 459.246,A -85,B 0,C 180,E1 -16636.088,E2 -16636.088} C_VEL
LIN {X 0,Y 291.144,Z 463.471,A -85,B 0,C 180,E1 -16638.158,E2 -16638.158} C_VEL
LIN {X 0,Y 290.267,Z 466.67,A -85,B 0,C 180,E1 -16640.241,E2 -16640.241} C_VEL
LIN {X 0,Y 289.583,Z 469.401,A -85,B 0,C 180,E1 -16643.029,E2 -16643.029} C_VEL
LIN {X 0,Y 289.477,Z 470.184,A -85,B 0,C 180,E1 -16644.507,E2 -16644.507} C_VEL
LIN {X 0,Y 289.484,Z 470.453,A -85,B 0,C 180,E1 -16645.822,E2 -16645.822} C_VEL
LIN {X 0,Y 289.503,Z 470.319,A -85,B 0,C 180,E1 -16647.216,E2 -16647.216} C_VEL
LIN {X 0,Y 289.793,Z 469.516,A -85,B 0,C 180,E1 -16649.998,E2 -16649.998} C_VEL
LIN {X 0,Y 289.563,Z 469.731,A -85,B 0,C 180,E1 -16652.781,E2 -16652.781} C_VEL
LIN {X 0,Y 289.5,Z 469.233,A -85,B 0,C 180,E1 -16654.175,E2 -16654.175} C_VEL
LIN {X 0,Y 289.515,Z 468.305,A -85,B 0,C 180,E1 -16655.571,E2 -16655.571} C_VEL
LIN {X 0,Y 289.821,Z 465.265,A -85,B 0,C 180,E1 -16658.364,E2 -16658.364} C_VEL
LIN {X 0,Y 290.34,Z 461.823,A -85,B 0,C 180,E1 -16660.458,E2 -16660.458} C_VEL
LIN {X 0,Y 291.153,Z 457.307,A -85,B 0,C 180,E1 -16662.546,E2 -16662.546} C_VEL
LIN {X 0,Y 292.813,Z 450.466,A -85,B 0,C 180,E1 -16664.951,E2 -16664.951} C_VEL
LIN {X 0,Y 294.503,Z 442.484,A -85,B 0,C 180,E1 -16667.152,E2 -16667.152} C_VEL
LIN {X 0,Y 296.44,Z 433.867,A -85,B 0,C 180,E1 -16669.024,E2 -16669.024} C_VEL
LIN {X 0,Y 298.783,Z 423.267,A -85,B 0,C 180,E1 -16670.839,E2 -16670.839} C_VEL
LIN {X 0,Y 300.895,Z 412.407,A -85,B 0,C 180,E1 -16672.304,E2 -16672.304} C_VEL
LIN {X 0,Y 302.97,Z 400.053,A -85,B 0,C 180,E1 -16673.586,E2 -16673.586} C_VEL
LIN {X 0,Y 304.76,Z 387.857,A -85,B 0,C 180,E1 -16674.524,E2 -16674.524} C_VEL
LIN {X 0,Y 306.153,Z 374.948,A -85,B 0,C 180,E1 -16675.22,E2 -16675.22} C_VEL
LIN {X 0,Y 306.94,Z 362.728,A -85,B 0,C 180,E1 -16675.65,E2 -16675.65} C_VEL
LIN {X 0,Y 308.63,Z 305.891,A -85,B 0,C 180,E1 -16677.009,E2 -16677.009} C_VEL
LIN {X 0,Y 305.963,Z 285.656,A -85,B 0,C 180,E1 -16677.873,E2 -16677.873} C_VEL
LIN {X 0,Y 301.833,Z 261.165,A -85,B 0,C 180,E1 -16679.064,E2 -16679.064} C_VEL
LIN {X 0,Y 295.572,Z 244.88,A -85,B 0,C 180,E1 -16680.366,E2 -16680.366} C_VEL
LIN {X 0,Y 293.037,Z 238.458,A -85,B 0,C 180,E1 -16680.986,E2 -16680.986} C_VEL
LIN {X 0,Y 291.514,Z 233.779,A -85,B 0,C 180,E1 -16681.419,E2 -16681.419} C_VEL
LIN {X 0,Y 291.44,Z 233.163,A -85,B 0,C 180,E1 -16681.635,E2 -16681.635} C_VEL
LIN {X 0,Y 291.35,Z 233.17,A -85,B 0,C 180,E1 -16685.373,E2 -16685.373} C_VEL
LIN {X 0,Y 291.357,Z 233.194,A -85,B 0,C 180,E1 -16687.249,E2 -16687.249} C_VEL
LIN {X 0,Y 291.289,Z 233.199,A -85,B 0,C 180,E1 -16691.588,E2 -16691.588} C_VEL
LIN {X 0,Y 291.276,Z 233.204,A -85,B 0,C 180,E1 -16695.595,E2 -16695.595} C_VEL
LIN {X 0,Y 291.292,Z 233.186,A -85,B 0,C 180,E1 -16699.351,E2 -16699.351} C_VEL
LIN {X 0,Y 291.383,Z 233.172,A -85,B 0,C 180,E1 -16702.916,E2 -16702.916} C_VEL
LIN {X 0,Y 291.336,Z 233.188,A -85,B 0,C 180,E1 -16706.301,E2 -16706.301} C_VEL
LIN {X 0,Y 291.327,Z 233.166,A -85,B 0,C 180,E1 -16710.278,E2 -16710.278} C_VEL
LIN {X 0,Y 291.349,Z 233.187,A -85,B 0,C 180,E1 -16714.266,E2 -16714.266} C_VEL
LIN {X 0,Y 291.354,Z 233.158,A -85,B 0,C 180,E1 -16717.298,E2 -16717.298} C_VEL
LIN {X 0,Y 291.384,Z 233.176,A -85,B 0,C 180,E1 -16720.265,E2 -16720.265} C_VEL
LIN {X 0,Y 291.489,Z 233.15,A -85,B 0,C 180,E1 -16724.665,E2 -16724.665} C_VEL
LIN {X 0,Y 291.52,Z 233.165,A -85,B 0,C 180,E1 -16728.88,E2 -16728.88} C_VEL
LIN {X 0,Y 291.642,Z 233.153,A -85,B 0,C 180,E1 -16731.687,E2 -16731.687} C_VEL
LIN {X 0,Y 291.59,Z 233.128,A -85,B 0,C 180,E1 -16734.468,E2 -16734.468} C_VEL
LIN {X 0,Y 291.865,Z 233.126,A -85,B 0,C 180,E1 -16738.621,E2 -16738.621} C_VEL
LIN {X 0,Y 291.872,Z 233.102,A -85,B 0,C 180,E1 -16741.38,E2 -16741.38} C_VEL
LIN {X 0,Y 291.726,Z 233.14,A -85,B 0,C 180,E1 -16746.919,E2 -16746.919} C_VEL
LIN {X 0,Y 291.567,Z 233.136,A -85,B 0,C 180,E1 -16749.714,E2 -16749.714} C_VEL
LIN {X 0,Y 291.508,Z 233.172,A -85,B 0,C 180,E1 -16753.951,E2 -16753.951} C_VEL
LIN {X 0,Y 291.435,Z 233.161,A -85,B 0,C 180,E1 -16758.271,E2 -16758.271} C_VEL
LIN {X 0,Y 291.365,Z 233.192,A -85,B 0,C 180,E1 -16761.212,E2 -16761.212} C_VEL
LIN {X 0,Y 291.393,Z 233.169,A -85,B 0,C 180,E1 -16764.206,E2 -16764.206} C_VEL
LIN {X 0,Y 291.415,Z 233.184,A -85,B 0,C 180,E1 -16767.273,E2 -16767.273} C_VEL
LIN {X 0,Y 291.328,Z 233.188,A -85,B 0,C 180,E1 -16770.438,E2 -16770.438} C_VEL
LIN {X 0,Y 291.339,Z 233.183,A -85,B 0,C 180,E1 -16773.7,E2 -16773.7} C_VEL
LIN {X 0,Y 291.371,Z 233.188,A -85,B 0,C 180,E1 -16777.256,E2 -16777.256} C_VEL
LIN {X 0,Y 291.328,Z 233.199,A -85,B 0,C 180,E1 -16780.644,E2 -16780.644} C_VEL
LIN {X 0,Y 291.32,Z 233.192,A -85,B 0,C 180,E1 -16784.941,E2 -16784.941} C_VEL
LIN {X 0,Y 291.314,Z 233.207,A -85,B 0,C 180,E1 -16785.113,E2 -16785.113} C_VEL
LIN {X 0,Y 292.187,Z 235.847,A -85,B 0,C 180,E1 -16785.317,E2 -16785.317} C_VEL
LIN {X 0,Y 294.01,Z 238.609,A -85,B 0,C 180,E1 -16785.656,E2 -16785.656} C_VEL
LIN {X 0,Y 303.276,Z 254.61,A -85,B 0,C 180,E1 -16787.346,E2 -16787.346} C_VEL
LIN {X 0,Y 310.372,Z 268.589,A -85,B 0,C 180,E1 -16788.59,E2 -16788.59} C_VEL
LIN {X 0,Y 307.932,Z 340.596,A -85,B 0,C 180,E1 -16790.281,E2 -16790.281} C_VEL
LIN {X 0,Y 307.107,Z 354.166,A -85,B 0,C 180,E1 -16790.842,E2 -16790.842} C_VEL
LIN {X 0,Y 306.045,Z 365.759,A -85,B 0,C 180,E1 -16791.57,E2 -16791.57} C_VEL
LIN {X 0,Y 304.59,Z 377.072,A -85,B 0,C 180,E1 -16792.516,E2 -16792.516} C_VEL
LIN {X 0,Y 302.859,Z 388.208,A -85,B 0,C 180,E1 -16793.721,E2 -16793.721} C_VEL
LIN {X 0,Y 300.783,Z 399.069,A -85,B 0,C 180,E1 -16795.208,E2 -16795.208} C_VEL
LIN {X 0,Y 298.765,Z 408.521,A -85,B 0,C 180,E1 -16796.846,E2 -16796.846} C_VEL
LIN {X 0,Y 296.905,Z 416.768,A -85,B 0,C 180,E1 -16798.619,E2 -16798.619} C_VEL
LIN {X 0,Y 294.946,Z 424.745,A -85,B 0,C 180,E1 -16800.761,E2 -16800.761} C_VEL
LIN {X 0,Y 293.328,Z 431.021,A -85,B 0,C 180,E1 -16802.922,E2 -16802.922} C_VEL
LIN {X 0,Y 292.07,Z 435.92,A -85,B 0,C 180,E1 -16805.098,E2 -16805.098} C_VEL
LIN {X 0,Y 291.074,Z 439.598,A -85,B 0,C 180,E1 -16807.276,E2 -16807.276} C_VEL
LIN {X 0,Y 290.507,Z 441.452,A -85,B 0,C 180,E1 -16808.724,E2 -16808.724} C_VEL
LIN {X 0,Y 289.897,Z 443.4,A -85,B 0,C 180,E1 -16810.995,E2 -16810.995} C_VEL
LIN {X 0,Y 289.532,Z 444.264,A -85,B 0,C 180,E1 -16813.067,E2 -16813.067} C_VEL
LIN {X 0,Y 289.401,Z 444.322,A -85,B 0,C 180,E1 -16814.508,E2 -16814.508} C_VEL
LIN {X 0,Y 289.396,Z 443.863,A -85,B 0,C 180,E1 -16816.268,E2 -16816.268} C_VEL
LIN {X 0,Y 289.435,Z 442.051,A -85,B 0,C 180,E1 -16818.8,E2 -16818.8} C_VEL
LIN {X 0,Y 289.684,Z 439.479,A -85,B 0,C 180,E1 -16820.928,E2 -16820.928} C_VEL
LIN {X 0,Y 290.155,Z 435.439,A -85,B 0,C 180,E1 -16823.262,E2 -16823.262} C_VEL
LIN {X 0,Y 290.549,Z 431.179,A -85,B 0,C 180,E1 -16825.145,E2 -16825.145} C_VEL
LIN {X 0,Y 291.417,Z 424.116,A -85,B 0,C 180,E1 -16827.583,E2 -16827.583} C_VEL
LIN {X 0,Y 292.415,Z 416.379,A -85,B 0,C 180,E1 -16829.657,E2 -16829.657} C_VEL
LIN {X 0,Y 293.688,Z 406.74,A -85,B 0,C 180,E1 -16831.716,E2 -16831.716} C_VEL
LIN {X 0,Y 295.001,Z 396.676,A -85,B 0,C 180,E1 -16833.416,E2 -16833.416} C_VEL
LIN {X 0,Y 296.354,Z 385.376,A -85,B 0,C 180,E1 -16834.934,E2 -16834.934} C_VEL
LIN {X 0,Y 297.452,Z 374.281,A -85,B 0,C 180,E1 -16836.105,E2 -16836.105} C_VEL
LIN {X 0,Y 298.23,Z 363.043,A -85,B 0,C 180,E1 -16837.023,E2 -16837.023} C_VEL
LIN {X 0,Y 299.016,Z 349.636,A -85,B 0,C 180,E1 -16837.811,E2 -16837.811} C_VEL
LIN {X 0,Y 299.555,Z 336.387,A -85,B 0,C 180,E1 -16838.293,E2 -16838.293} C_VEL
LIN {X 0,Y 301.302,Z 260.856,A -85,B 0,C 180,E1 -16840.07,E2 -16840.07} C_VEL
LIN {X 0,Y 300.228,Z 255.062,A -85,B 0,C 180,E1 -16840.29,E2 -16840.29} C_VEL
LIN {X 0,Y 291.669,Z 234.025,A -85,B 0,C 180,E1 -16841.446,E2 -16841.446} C_VEL
LIN {X 0,Y 291.526,Z 233.171,A -85,B 0,C 180,E1 -16841.499,E2 -16841.499} C_VEL
LIN {X 0,Y 291.561,Z 233.165,A -85,B 0,C 180,E1 -16845.377,E2 -16845.377} C_VEL
LIN {X 0,Y 291.457,Z 233.18,A -85,B 0,C 180,E1 -16849.876,E2 -16849.876} C_VEL
LIN {X 0,Y 291.352,Z 233.195,A -85,B 0,C 180,E1 -16854.211,E2 -16854.211} C_VEL
LIN {X 0,Y 291.335,Z 233.192,A -85,B 0,C 180,E1 -16857.282,E2 -16857.282} C_VEL
LIN {X 0,Y 291.308,Z 233.194,A -85,B 0,C 180,E1 -16860.442,E2 -16860.442} C_VEL
LIN {X 0,Y 291.35,Z 233.195,A -85,B 0,C 180,E1 -16863.699,E2 -16863.699} C_VEL
LIN {X 0,Y 291.358,Z 233.189,A -85,B 0,C 180,E1 -16867.248,E2 -16867.248} C_VEL
LIN {X 0,Y 291.306,Z 233.196,A -85,B 0,C 180,E1 -16870.649,E2 -16870.649} C_VEL
LIN {X 0,Y 291.288,Z 233.196,A -85,B 0,C 180,E1 -16874.404,E2 -16874.404} C_VEL
LIN {X 0,Y 291.3,Z 233.196,A -85,B 0,C 180,E1 -16878.412,E2 -16878.412} C_VEL
LIN {X 0,Y 291.393,Z 233.182,A -85,B 0,C 180,E1 -16882.917,E2 -16882.917} C_VEL
LIN {X 0,Y 291.349,Z 233.19,A -85,B 0,C 180,E1 -16886.302,E2 -16886.302} C_VEL
LIN {X 0,Y 291.344,Z 233.187,A -85,B 0,C 180,E1 -16890.278,E2 -16890.278} C_VEL
LIN {X 0,Y 291.325,Z 233.186,A -85,B 0,C 180,E1 -16890.882,E2 -16890.882} C_VEL
LIN {X 0,Y 290.645,Z 233.271,A -85,B 0,C 180,E1 -16891.651,E2 -16891.651} C_VEL
LIN {X 0,Y 287.8,Z 233.627,A -85,B 0,C 180,E1 -16892.857,E2 -16892.857} C_VEL
LIN {X 0,Y 284.979,Z 233.977,A -85,B 0,C 180,E1 -16894.086,E2 -16894.086} C_VEL
LIN {X 0,Y 284.365,Z 234.057,A -85,B 0,C 180,E1 -16894.88,E2 -16894.88} C_VEL
LIN {X 0,Y 284.4,Z 234.056,A -85,B 0,C 180,E1 -16895.188,E2 -16895.188} C_VEL
LIN {X 0,Y 290.949,Z 259.486,A -85,B 0,C 180,E1 -16896.452,E2 -16896.452} C_VEL
LIN {X 0,Y 291.345,Z 263.885,A -85,B 0,C 180,E1 -16896.635,E2 -16896.635} C_VEL
LIN {X 0,Y 288.368,Z 342.44,A -85,B 0,C 180,E1 -16899.584,E2 -16899.584} C_VEL
LIN {X 0,Y 287.851,Z 356.343,A -85,B 0,C 180,E1 -16900.384,E2 -16900.384} C_VEL
LIN {X 0,Y 287.128,Z 369.658,A -85,B 0,C 180,E1 -16901.445,E2 -16901.445} C_VEL
LIN {X 0,Y 286.308,Z 381.649,A -85,B 0,C 180,E1 -16902.684,E2 -16902.684} C_VEL
LIN {X 0,Y 285.454,Z 392.568,A -85,B 0,C 180,E1 -16904.088,E2 -16904.088} C_VEL
LIN {X 0,Y 284.716,Z 402.804,A -85,B 0,C 180,E1 -16905.709,E2 -16905.709} C_VEL
LIN {X 0,Y 284.002,Z 412.101,A -85,B 0,C 180,E1 -16907.494,E2 -16907.494} C_VEL
LIN {X 0,Y 283.49,Z 419.8,A -85,B 0,C 180,E1 -16909.284,E2 -16909.284} C_VEL
LIN {X 0,Y 282.997,Z 427.33,A -85,B 0,C 180,E1 -16911.43,E2 -16911.43} C_VEL
LIN {X 0,Y 282.673,Z 433.526,A -85,B 0,C 180,E1 -16913.647,E2 -16913.647} C_VEL
LIN {X 0,Y 282.559,Z 438.085,A -85,B 0,C 180,E1 -16915.72,E2 -16915.72} C_VEL
LIN {X 0,Y 282.482,Z 441.645,A -85,B 0,C 180,E1 -16917.861,E2 -16917.861} C_VEL
LIN {X 0,Y 282.517,Z 444.162,A -85,B 0,C 180,E1 -16920,E2 -16920} C_VEL
LIN {X 0,Y 282.68,Z 445.298,A -85,B 0,C 180,E1 -16921.424,E2 -16921.424} C_VEL
LIN {X 0,Y 282.937,Z 446.007,A -85,B 0,C 180,E1 -16922.847,E2 -16922.847} C_VEL
LIN {X 0,Y 283.334,Z 446.254,A -85,B 0,C 180,E1 -16924.267,E2 -16924.267} C_VEL
LIN {X 0,Y 283.824,Z 446.094,A -85,B 0,C 180,E1 -16925.684,E2 -16925.684} C_VEL
LIN {X 0,Y 284.176,Z 445.557,A -85,B 0,C 180,E1 -16927.103,E2 -16927.103} C_VEL
LIN {X 0,Y 284.614,Z 444.605,A -85,B 0,C 180,E1 -16928.52,E2 -16928.52} C_VEL
LIN {X 0,Y 286.524,Z 441.545,A -85,B 0,C 180,E1 -16931.139,E2 -16931.139} C_VEL
LIN {X 0,Y 288.387,Z 437.656,A -85,B 0,C 180,E1 -16933.386,E2 -16933.386} C_VEL
LIN {X 0,Y 290.422,Z 432.931,A -85,B 0,C 180,E1 -16935.438,E2 -16935.438} C_VEL
LIN {X 0,Y 292.828,Z 426.994,A -85,B 0,C 180,E1 -16937.458,E2 -16937.458} C_VEL
LIN {X 0,Y 295.56,Z 419.636,A -85,B 0,C 180,E1 -16939.445,E2 -16939.445} C_VEL
LIN {X 0,Y 298.739,Z 410.523,A -85,B 0,C 180,E1 -16941.386,E2 -16941.386} C_VEL
LIN {X 0,Y 301.942,Z 400.33,A -85,B 0,C 180,E1 -16943.128,E2 -16943.128} C_VEL
LIN {X 0,Y 305.348,Z 387.711,A -85,B 0,C 180,E1 -16944.837,E2 -16944.837} C_VEL
LIN {X 0,Y 308.454,Z 374.5,A -85,B 0,C 180,E1 -16946.196,E2 -16946.196} C_VEL
LIN {X 0,Y 310.941,Z 361.405,A -85,B 0,C 180,E1 -16947.238,E2 -16947.238} C_VEL
LIN {X 0,Y 313.103,Z 347.679,A -85,B 0,C 180,E1 -16948.032,E2 -16948.032} C_VEL
LIN {X 0,Y 320.48,Z 291.283,A -85,B 0,C 180,E1 -16950.381,E2 -16950.381} C_VEL
LIN {X 0,Y 317.424,Z 285.104,A -85,B 0,C 180,E1 -16951.838,E2 -16951.838} C_VEL
LIN {X 0,Y 313.642,Z 278.597,A -85,B 0,C 180,E1 -16953.875,E2 -16953.875} C_VEL
LIN {X 0,Y 310.899,Z 274.545,A -85,B 0,C 180,E1 -16955.625,E2 -16955.625} C_VEL
LIN {X 0,Y 308.356,Z 270.938,A -85,B 0,C 180,E1 -16957.704,E2 -16957.704} C_VEL
LIN {X 0,Y 305.63,Z 268.01,A -85,B 0,C 180,E1 -16961.079,E2 -16961.079} C_VEL
LIN {X 0,Y 305.045,Z 267.617,A -85,B 0,C 180,E1 -16962.5,E2 -16962.5} C_VEL
LIN {X 0,Y 304.815,Z 268.207,A -85,B 0,C 180,E1 -16965.225,E2 -16965.225} C_VEL
LIN {X 0,Y 305.789,Z 270.172,A -85,B 0,C 180,E1 -16967.845,E2 -16967.845} C_VEL
LIN {X 0,Y 308.583,Z 276.022,A -85,B 0,C 180,E1 -16971.278,E2 -16971.278} C_VEL
LIN {X 0,Y 309.766,Z 278.292,A -85,B 0,C 180,E1 -16972.272,E2 -16972.272} C_VEL
LIN {X 0,Y 312.45,Z 283.969,A -85,B 0,C 180,E1 -16974.208,E2 -16974.208} C_VEL
LIN {X 0,Y 314.78,Z 289.387,A -85,B 0,C 180,E1 -16975.654,E2 -16975.654} C_VEL
LIN {X 0,Y 317.122,Z 295.374,A -85,B 0,C 180,E1 -16976.961,E2 -16976.961} C_VEL
LIN {X 0,Y 317.494,Z 297.772,A -85,B 0,C 180,E1 -16977.279,E2 -16977.279} C_VEL
LIN {X 0,Y 318.303,Z 309.893,A -85,B 0,C 180,E1 -16978.479,E2 -16978.479} C_VEL
LIN {X 0,Y 318.198,Z 313.804,A -85,B 0,C 180,E1 -16978.746,E2 -16978.746} C_VEL
LIN {X 0,Y 311.399,Z 367.126,A -85,B 0,C 180,E1 -16980.971,E2 -16980.971} C_VEL
LIN {X 0,Y 308.99,Z 380.619,A -85,B 0,C 180,E1 -16981.744,E2 -16981.744} C_VEL
LIN {X 0,Y 306.192,Z 393.027,A -85,B 0,C 180,E1 -16982.672,E2 -16982.672} C_VEL
LIN {X 0,Y 303.116,Z 405.243,A -85,B 0,C 180,E1 -16983.861,E2 -16983.861} C_VEL
LIN {X 0,Y 299.587,Z 417.562,A -85,B 0,C 180,E1 -16985.391,E2 -16985.391} C_VEL
LIN {X 0,Y 296.502,Z 427.683,A -85,B 0,C 180,E1 -16986.976,E2 -16986.976} C_VEL
LIN {X 0,Y 293.187,Z 437.67,A -85,B 0,C 180,E1 -16988.925,E2 -16988.925} C_VEL
LIN {X 0,Y 290.043,Z 446.686,A -85,B 0,C 180,E1 -16991.129,E2 -16991.129} C_VEL
LIN {X 0,Y 288.045,Z 452.675,A -85,B 0,C 180,E1 -16992.974,E2 -16992.974} C_VEL
LIN {X 0,Y 286.165,Z 458.153,A -85,B 0,C 180,E1 -16995.055,E2 -16995.055} C_VEL
LIN {X 0,Y 284.564,Z 462.524,A -85,B 0,C 180,E1 -16997.156,E2 -16997.156} C_VEL
LIN {X 0,Y 283.822,Z 464.829,A -85,B 0,C 180,E1 -16998.573,E2 -16998.573} C_VEL
LIN {X 0,Y 282.807,Z 468.185,A -85,B 0,C 180,E1 -17001.423,E2 -17001.423} C_VEL
LIN {X 0,Y 282.508,Z 469.233,A -85,B 0,C 180,E1 -17002.853,E2 -17002.853} C_VEL
LIN {X 0,Y 282.381,Z 469.91,A -85,B 0,C 180,E1 -17004.583,E2 -17004.583} C_VEL
LIN {X 0,Y 282.429,Z 469.817,A -85,B 0,C 180,E1 -17007.146,E2 -17007.146} C_VEL
LIN {X 0,Y 282.616,Z 468.832,A -85,B 0,C 180,E1 -17009.286,E2 -17009.286} C_VEL
LIN {X 0,Y 282.527,Z 469.489,A -85,B 0,C 180,E1 -17011.424,E2 -17011.424} C_VEL
LIN {X 0,Y 282.484,Z 469.429,A -85,B 0,C 180,E1 -17012.851,E2 -17012.851} C_VEL
LIN {X 0,Y 282.417,Z 468.25,A -85,B 0,C 180,E1 -17015.494,E2 -17015.494} C_VEL
LIN {X 0,Y 282.503,Z 466.779,A -85,B 0,C 180,E1 -17017.144,E2 -17017.144} C_VEL
LIN {X 0,Y 282.926,Z 464.059,A -85,B 0,C 180,E1 -17019.29,E2 -17019.29} C_VEL
LIN {X 0,Y 283.584,Z 460.331,A -85,B 0,C 180,E1 -17021.434,E2 -17021.434} C_VEL
LIN {X 0,Y 284.664,Z 455.491,A -85,B 0,C 180,E1 -17023.563,E2 -17023.563} C_VEL
LIN {X 0,Y 286.191,Z 449.397,A -85,B 0,C 180,E1 -17025.67,E2 -17025.67} C_VEL
LIN {X 0,Y 287.959,Z 441.487,A -85,B 0,C 180,E1 -17027.854,E2 -17027.854} C_VEL
LIN {X 0,Y 290.139,Z 432.366,A -85,B 0,C 180,E1 -17029.822,E2 -17029.822} C_VEL
LIN {X 0,Y 292.402,Z 422.589,A -85,B 0,C 180,E1 -17031.501,E2 -17031.501} C_VEL
LIN {X 0,Y 294.641,Z 411.611,A -85,B 0,C 180,E1 -17032.989,E2 -17032.989} C_VEL
LIN {X 0,Y 296.522,Z 400.881,A -85,B 0,C 180,E1 -17034.131,E2 -17034.131} C_VEL
LIN {X 0,Y 298.337,Z 389.054,A -85,B 0,C 180,E1 -17035.088,E2 -17035.088} C_VEL
LIN {X 0,Y 299.901,Z 376.084,A -85,B 0,C 180,E1 -17035.83,E2 -17035.83} C_VEL
LIN {X 0,Y 300.789,Z 363.348,A -85,B 0,C 180,E1 -17036.307,E2 -17036.307} C_VEL
LIN {X 0,Y 302.557,Z 306.486,A -85,B 0,C 180,E1 -17037.699,E2 -17037.699} C_VEL
LIN {X 0,Y 299.506,Z 283.729,A -85,B 0,C 180,E1 -17038.717,E2 -17038.717} C_VEL
LIN {X 0,Y 296.124,Z 263.72,A -85,B 0,C 180,E1 -17039.73,E2 -17039.73} C_VEL
LIN {X 0,Y 289.963,Z 247.723,A -85,B 0,C 180,E1 -17041.054,E2 -17041.054} C_VEL
LIN {X 0,Y 286.159,Z 237.912,A -85,B 0,C 180,E1 -17042.008,E2 -17042.008} C_VEL
LIN {X 0,Y 284.63,Z 235.316,A -85,B 0,C 180,E1 -17042.358,E2 -17042.358} C_VEL
LIN {X 0,Y 284.319,Z 234.034,A -85,B 0,C 180,E1 -17042.503,E2 -17042.503} C_VEL
LIN {X 0,Y 284.319,Z 234.065,A -85,B 0,C 180,E1 -17046.386,E2 -17046.386} C_VEL
LIN {X 0,Y 284.248,Z 234.07,A -85,B 0,C 180,E1 -17050.002,E2 -17050.002} C_VEL
LIN {X 0,Y 284.227,Z 234.07,A -85,B 0,C 180,E1 -17054.187,E2 -17054.187} C_VEL
LIN {X 0,Y 284.232,Z 234.06,A -85,B 0,C 180,E1 -17058.117,E2 -17058.117} C_VEL
LIN {X 0,Y 284.301,Z 234.064,A -85,B 0,C 180,E1 -17062.281,E2 -17062.281} C_VEL
LIN {X 0,Y 284.299,Z 234.052,A -85,B 0,C 180,E1 -17065.35,E2 -17065.35} C_VEL
LIN {X 0,Y 284.27,Z 234.061,A -85,B 0,C 180,E1 -17068.723,E2 -17068.723} C_VEL
LIN {X 0,Y 284.253,Z 234.053,A -85,B 0,C 180,E1 -17071.981,E2 -17071.981} C_VEL
LIN {X 0,Y 284.312,Z 234.05,A -85,B 0,C 180,E1 -17076.147,E2 -17076.147} C_VEL
LIN {X 0,Y 284.325,Z 234.05,A -85,B 0,C 180,E1 -17079.928,E2 -17079.928} C_VEL
LIN {X 0,Y 284.437,Z 234.03,A -85,B 0,C 180,E1 -17084.493,E2 -17084.493} C_VEL
LIN {X 0,Y 284.473,Z 234.039,A -85,B 0,C 180,E1 -17088.601,E2 -17088.601} C_VEL
LIN {X 0,Y 284.599,Z 234.03,A -85,B 0,C 180,E1 -17091.48,E2 -17091.48} C_VEL
LIN {X 0,Y 284.56,Z 234.003,A -85,B 0,C 180,E1 -17094.331,E2 -17094.331} C_VEL
LIN {X 0,Y 284.832,Z 234.002,A -85,B 0,C 180,E1 -17098.586,E2 -17098.586} C_VEL
LIN {X 0,Y 284.838,Z 233.977,A -85,B 0,C 180,E1 -17101.414,E2 -17101.414} C_VEL
LIN {X 0,Y 284.678,Z 234.017,A -85,B 0,C 180,E1 -17107.091,E2 -17107.091} C_VEL
LIN {X 0,Y 284.511,Z 234.013,A -85,B 0,C 180,E1 -17109.958,E2 -17109.958} C_VEL
LIN {X 0,Y 284.456,Z 234.048,A -85,B 0,C 180,E1 -17114.305,E2 -17114.305} C_VEL
LIN {X 0,Y 284.375,Z 234.045,A -85,B 0,C 180,E1 -17118.741,E2 -17118.741} C_VEL
LIN {X 0,Y 284.318,Z 234.063,A -85,B 0,C 180,E1 -17121.764,E2 -17121.764} C_VEL
LIN {X 0,Y 284.34,Z 234.052,A -85,B 0,C 180,E1 -17124.847,E2 -17124.847} C_VEL
LIN {X 0,Y 284.322,Z 234.061,A -85,B 0,C 180,E1 -17128.012,E2 -17128.012} C_VEL
LIN {X 0,Y 284.288,Z 234.072,A -85,B 0,C 180,E1 -17131.276,E2 -17131.276} C_VEL
LIN {X 0,Y 284.336,Z 234.063,A -85,B 0,C 180,E1 -17135.35,E2 -17135.35} C_VEL
LIN {X 0,Y 284.307,Z 234.062,A -85,B 0,C 180,E1 -17138.17,E2 -17138.17} C_VEL
LIN {X 0,Y 284.264,Z 234.069,A -85,B 0,C 180,E1 -17142.126,E2 -17142.126} C_VEL
LIN {X 0,Y 284.289,Z 234.237,A -85,B 0,C 180,E1 -17144.107,E2 -17144.107} C_VEL
LIN {X 0,Y 285.197,Z 236.848,A -85,B 0,C 180,E1 -17144.326,E2 -17144.326} C_VEL
LIN {X 0,Y 286.824,Z 239.1,A -85,B 0,C 180,E1 -17144.639,E2 -17144.639} C_VEL
LIN {X 0,Y 297.369,Z 257.125,A -85,B 0,C 180,E1 -17146.655,E2 -17146.655} C_VEL
LIN {X 0,Y 304.355,Z 270.907,A -85,B 0,C 180,E1 -17147.935,E2 -17147.935} C_VEL
LIN {X 0,Y 301.788,Z 341.908,A -85,B 0,C 180,E1 -17149.635,E2 -17149.635} C_VEL
LIN {X 0,Y 300.898,Z 355.337,A -85,B 0,C 180,E1 -17150.218,E2 -17150.218} C_VEL
LIN {X 0,Y 299.658,Z 367.705,A -85,B 0,C 180,E1 -17151.037,E2 -17151.037} C_VEL
LIN {X 0,Y 297.882,Z 380.365,A -85,B 0,C 180,E1 -17152.165,E2 -17152.165} C_VEL
LIN {X 0,Y 295.866,Z 392.167,A -85,B 0,C 180,E1 -17153.571,E2 -17153.571} C_VEL
LIN {X 0,Y 293.644,Z 402.702,A -85,B 0,C 180,E1 -17155.153,E2 -17155.153} C_VEL
LIN {X 0,Y 291.725,Z 411.253,A -85,B 0,C 180,E1 -17156.767,E2 -17156.767} C_VEL
LIN {X 0,Y 289.809,Z 419.033,A -85,B 0,C 180,E1 -17158.577,E2 -17158.577} C_VEL
LIN {X 0,Y 287.833,Z 426.581,A -85,B 0,C 180,E1 -17160.771,E2 -17160.771} C_VEL
LIN {X 0,Y 286.179,Z 432.562,A -85,B 0,C 180,E1 -17162.98,E2 -17162.98} C_VEL
LIN {X 0,Y 284.925,Z 437.174,A -85,B 0,C 180,E1 -17165.21,E2 -17165.21} C_VEL
LIN {X 0,Y 284.212,Z 439.556,A -85,B 0,C 180,E1 -17166.695,E2 -17166.695} C_VEL
LIN {X 0,Y 283.603,Z 441.484,A -85,B 0,C 180,E1 -17168.18,E2 -17168.18} C_VEL
LIN {X 0,Y 282.853,Z 443.725,A -85,B 0,C 180,E1 -17170.768,E2 -17170.768} C_VEL
LIN {X 0,Y 282.514,Z 444.513,A -85,B 0,C 180,E1 -17172.633,E2 -17172.633} C_VEL
LIN {X 0,Y 282.354,Z 444.67,A -85,B 0,C 180,E1 -17174.111,E2 -17174.111} C_VEL
LIN {X 0,Y 282.308,Z 444.185,A -85,B 0,C 180,E1 -17176.146,E2 -17176.146} C_VEL
LIN {X 0,Y 282.343,Z 442.607,A -85,B 0,C 180,E1 -17178.515,E2 -17178.515} C_VEL
LIN {X 0,Y 282.457,Z 441.053,A -85,B 0,C 180,E1 -17179.971,E2 -17179.971} C_VEL
LIN {X 0,Y 282.833,Z 437.916,A -85,B 0,C 180,E1 -17182.147,E2 -17182.147} C_VEL
LIN {X 0,Y 283.279,Z 433.718,A -85,B 0,C 180,E1 -17184.306,E2 -17184.306} C_VEL
LIN {X 0,Y 284.026,Z 427.343,A -85,B 0,C 180,E1 -17186.81,E2 -17186.81} C_VEL
LIN {X 0,Y 284.888,Z 420.338,A -85,B 0,C 180,E1 -17188.941,E2 -17188.941} C_VEL
LIN {X 0,Y 286.106,Z 411.595,A -85,B 0,C 180,E1 -17191.057,E2 -17191.057} C_VEL
LIN {X 0,Y 287.335,Z 402.633,A -85,B 0,C 180,E1 -17192.805,E2 -17192.805} C_VEL
LIN {X 0,Y 288.652,Z 392.684,A -85,B 0,C 180,E1 -17194.365,E2 -17194.365} C_VEL
LIN {X 0,Y 289.881,Z 381.888,A -85,B 0,C 180,E1 -17195.723,E2 -17195.723} C_VEL
LIN {X 0,Y 290.845,Z 371.41,A -85,B 0,C 180,E1 -17196.77,E2 -17196.77} C_VEL
LIN {X 0,Y 291.803,Z 359.181,A -85,B 0,C 180,E1 -17197.701,E2 -17197.701} C_VEL
LIN {X 0,Y 292.509,Z 345.912,A -85,B 0,C 180,E1 -17198.396,E2 -17198.396} C_VEL
LIN {X 0,Y 292.942,Z 331.482,A -85,B 0,C 180,E1 -17198.843,E2 -17198.843} C_VEL
LIN {X 0,Y 294.58,Z 261.382,A -85,B 0,C 180,E1 -17200.526,E2 -17200.526} C_VEL
LIN {X 0,Y 293.697,Z 257.058,A -85,B 0,C 180,E1 -17200.7,E2 -17200.7} C_VEL
LIN {X 0,Y 284.622,Z 234.887,A -85,B 0,C 180,E1 -17201.97,E2 -17201.97} C_VEL
LIN {X 0,Y 284.468,Z 234.051,A -85,B 0,C 180,E1 -17202.034,E2 -17202.034} C_VEL
LIN {X 0,Y 284.494,Z 234.046,A -85,B 0,C 180,E1 -17205.769,E2 -17205.769} C_VEL
LIN {X 0,Y 284.383,Z 234.062,A -85,B 0,C 180,E1 -17210.243,E2 -17210.243} C_VEL
LIN {X 0,Y 284.316,Z 234.069,A -85,B 0,C 180,E1 -17213.849,E2 -17213.849} C_VEL
LIN {X 0,Y 284.266,Z 234.077,A -85,B 0,C 180,E1 -17218.019,E2 -17218.019} C_VEL
LIN {X 0,Y 284.284,Z 234.069,A -85,B 0,C 180,E1 -17221.277,E2 -17221.277} C_VEL
LIN {X 0,Y 284.343,Z 234.065,A -85,B 0,C 180,E1 -17225.347,E2 -17225.347} C_VEL
LIN {X 0,Y 284.301,Z 234.07,A -85,B 0,C 180,E1 -17228.172,E2 -17228.172} C_VEL
LIN {X 0,Y 284.242,Z 234.072,A -85,B 0,C 180,E1 -17232.117,E2 -17232.117} C_VEL
LIN {X 0,Y 284.244,Z 234.076,A -85,B 0,C 180,E1 -17236.186,E2 -17236.186} C_VEL
LIN {X 0,Y 284.262,Z 234.069,A -85,B 0,C 180,E1 -17240.037,E2 -17240.037} C_VEL
LIN {X 0,Y 284.325,Z 234.065,A -85,B 0,C 180,E1 -17243.612,E2 -17243.612} C_VEL
LIN {X 0,Y 284.312,Z 234.069,A -85,B 0,C 180,E1 -17247.191,E2 -17247.191} C_VEL
LIN {X 0,Y 284.28,Z 234.062,A -85,B 0,C 180,E1 -17250.866,E2 -17250.866} C_VEL
LIN {X 0,Y 284.365,Z 234.057,A -85,B 0,C 180,E1 -17254.88,E2 -17254.88} C_VEL
LIN {X 0,Y 285.274,Z 234.298,A -85,B 0,C 180,E1 -17255.172,E2 -17255.172} C_VEL
LIN {X 0,Y 287.863,Z 235.073,A -85,B 0,C 180,E1 -17255.387,E2 -17255.387} C_VEL
LIN {X 0,Y 294.259,Z 237.966,A -85,B 0,C 180,E1 -17255.753,E2 -17255.753} C_VEL
LIN {X 0,Y 297.806,Z 240.897,A -85,B 0,C 180,E1 -17256.023,E2 -17256.023} C_VEL
LIN {X 0,Y 299.388,Z 243.516,A -85,B 0,C 180,E1 -17256.184,E2 -17256.184} C_VEL
LIN {X 0,Y 299.692,Z 246.3,A -85,B 0,C 180,E1 -17256.28,E2 -17256.28} C_VEL
LIN {X 0,Y 298.639,Z 249.148,A -85,B 0,C 180,E1 -17256.292,E2 -17256.292} C_VEL
LIN {X 0,Y 296.106,Z 252.165,A -85,B 0,C 180,E1 -17256.283,E2 -17256.283} C_VEL
LIN {X 0,Y 286.632,Z 259.986,A -85,B 0,C 180,E1 -17256.283,E2 -17256.283} C_VEL
LIN {X 0,Y 284.648,Z 263.308,A -85,B 0,C 180,E1 -17256.36,E2 -17256.36} C_VEL
LIN {X 0,Y 284.342,Z 264.801,A -85,B 0,C 180,E1 -17256.41,E2 -17256.41} C_VEL
LIN {X 0,Y 281.283,Z 343.284,A -85,B 0,C 180,E1 -17259.477,E2 -17259.477} C_VEL
LIN {X 0,Y 280.696,Z 357.648,A -85,B 0,C 180,E1 -17260.339,E2 -17260.339} C_VEL
LIN {X 0,Y 280.054,Z 369.739,A -85,B 0,C 180,E1 -17261.339,E2 -17261.339} C_VEL
LIN {X 0,Y 279.134,Z 383.096,A -85,B 0,C 180,E1 -17262.766,E2 -17262.766} C_VEL
LIN {X 0,Y 278.18,Z 395.202,A -85,B 0,C 180,E1 -17264.429,E2 -17264.429} C_VEL
LIN {X 0,Y 277.487,Z 404.989,A -85,B 0,C 180,E1 -17266.077,E2 -17266.077} C_VEL
LIN {X 0,Y 276.753,Z 413.936,A -85,B 0,C 180,E1 -17267.906,E2 -17267.906} C_VEL
LIN {X 0,Y 276.166,Z 422.698,A -85,B 0,C 180,E1 -17270.108,E2 -17270.108} C_VEL
LIN {X 0,Y 275.748,Z 429.751,A -85,B 0,C 180,E1 -17272.31,E2 -17272.31} C_VEL
LIN {X 0,Y 275.536,Z 434.493,A -85,B 0,C 180,E1 -17274.144,E2 -17274.144} C_VEL
LIN {X 0,Y 275.463,Z 439.06,A -85,B 0,C 180,E1 -17276.343,E2 -17276.343} C_VEL
LIN {X 0,Y 275.389,Z 442.469,A -85,B 0,C 180,E1 -17278.537,E2 -17278.537} C_VEL
LIN {X 0,Y 275.432,Z 444.169,A -85,B 0,C 180,E1 -17280,E2 -17280} C_VEL
LIN {X 0,Y 275.595,Z 445.408,A -85,B 0,C 180,E1 -17281.461,E2 -17281.461} C_VEL
LIN {X 0,Y 275.859,Z 446.237,A -85,B 0,C 180,E1 -17282.92,E2 -17282.92} C_VEL
LIN {X 0,Y 276.268,Z 446.659,A -85,B 0,C 180,E1 -17284.377,E2 -17284.377} C_VEL
LIN {X 0,Y 276.77,Z 446.626,A -85,B 0,C 180,E1 -17285.829,E2 -17285.829} C_VEL
LIN {X 0,Y 277.652,Z 445.383,A -85,B 0,C 180,E1 -17288.735,E2 -17288.735} C_VEL
LIN {X 0,Y 278.731,Z 444.11,A -85,B 0,C 180,E1 -17290.166,E2 -17290.166} C_VEL
LIN {X 0,Y 280.374,Z 441.391,A -85,B 0,C 180,E1 -17292.302,E2 -17292.302} C_VEL
LIN {X 0,Y 282.309,Z 437.655,A -85,B 0,C 180,E1 -17294.415,E2 -17294.415} C_VEL
LIN {X 0,Y 284.607,Z 432.82,A -85,B 0,C 180,E1 -17296.498,E2 -17296.498} C_VEL
LIN {X 0,Y 287.221,Z 426.776,A -85,B 0,C 180,E1 -17298.548,E2 -17298.548} C_VEL
LIN {X 0,Y 290.247,Z 419.274,A -85,B 0,C 180,E1 -17300.554,E2 -17300.554} C_VEL
LIN {X 0,Y 293.652,Z 410.094,A -85,B 0,C 180,E1 -17302.515,E2 -17302.515} C_VEL
LIN {X 0,Y 297.131,Z 399.692,A -85,B 0,C 180,E1 -17304.266,E2 -17304.266} C_VEL
LIN {X 0,Y 300.423,Z 388.251,A -85,B 0,C 180,E1 -17305.83,E2 -17305.83} C_VEL
LIN {X 0,Y 303.764,Z 375.167,A -85,B 0,C 180,E1 -17307.19,E2 -17307.19} C_VEL
LIN {X 0,Y 306.394,Z 362.297,A -85,B 0,C 180,E1 -17308.235,E2 -17308.235} C_VEL
LIN {X 0,Y 308.689,Z 348.969,A -85,B 0,C 180,E1 -17309.027,E2 -17309.027} C_VEL
LIN {X 0,Y 316.243,Z 294.937,A -85,B 0,C 180,E1 -17311.336,E2 -17311.336} C_VEL
LIN {X 0,Y 313.93,Z 290.197,A -85,B 0,C 180,E1 -17312.554,E2 -17312.554} C_VEL
LIN {X 0,Y 311.509,Z 285.798,A -85,B 0,C 180,E1 -17313.952,E2 -17313.952} C_VEL
LIN {X 0,Y 308.591,Z 281.063,A -85,B 0,C 180,E1 -17315.927,E2 -17315.927} C_VEL
LIN {X 0,Y 306.366,Z 277.706,A -85,B 0,C 180,E1 -17317.854,E2 -17317.854} C_VEL
LIN {X 0,Y 303.785,Z 274.821,A -85,B 0,C 180,E1 -17321.224,E2 -17321.224} C_VEL
LIN {X 0,Y 303.377,Z 274.51,A -85,B 0,C 180,E1 -17322.207,E2 -17322.207} C_VEL
LIN {X 0,Y 303.02,Z 274.906,A -85,B 0,C 180,E1 -17324.828,E2 -17324.828} C_VEL
LIN {X 0,Y 303.859,Z 276.854,A -85,B 0,C 180,E1 -17327.58,E2 -17327.58} C_VEL
LIN {X 0,Y 306.333,Z 282.575,A -85,B 0,C 180,E1 -17330.963,E2 -17330.963} C_VEL
LIN {X 0,Y 307.322,Z 284.599,A -85,B 0,C 180,E1 -17331.868,E2 -17331.868} C_VEL
LIN {X 0,Y 309.621,Z 289.874,A -85,B 0,C 180,E1 -17333.691,E2 -17333.691} C_VEL
LIN {X 0,Y 311.788,Z 295.306,A -85,B 0,C 180,E1 -17335.158,E2 -17335.158} C_VEL
LIN {X 0,Y 313.629,Z 300.381,A -85,B 0,C 180,E1 -17336.296,E2 -17336.296} C_VEL
LIN {X 0,Y 314.127,Z 310.846,A -85,B 0,C 180,E1 -17337.378,E2 -17337.378} C_VEL
LIN {X 0,Y 314.095,Z 315.069,A -85,B 0,C 180,E1 -17337.723,E2 -17337.723} C_VEL
LIN {X 0,Y 307.057,Z 366.391,A -85,B 0,C 180,E1 -17339.906,E2 -17339.906} C_VEL
LIN {X 0,Y 304.386,Z 380.334,A -85,B 0,C 180,E1 -17340.71,E2 -17340.71} C_VEL
LIN {X 0,Y 301.446,Z 392.561,A -85,B 0,C 180,E1 -17341.637,E2 -17341.637} C_VEL
LIN {X 0,Y 298.175,Z 404.703,A -85,B 0,C 180,E1 -17342.826,E2 -17342.826} C_VEL
LIN {X 0,Y 294.438,Z 416.931,A -85,B 0,C 180,E1 -17344.364,E2 -17344.364} C_VEL
LIN {X 0,Y 291.413,Z 426.073,A -85,B 0,C 180,E1 -17345.794,E2 -17345.794} C_VEL
LIN {X 0,Y 288.405,Z 434.708,A -85,B 0,C 180,E1 -17347.429,E2 -17347.429} C_VEL
LIN {X 0,Y 284.889,Z 444.035,A -85,B 0,C 180,E1 -17349.625,E2 -17349.625} C_VEL
LIN {X 0,Y 282,Z 451.493,A -85,B 0,C 180,E1 -17351.847,E2 -17351.847} C_VEL
LIN {X 0,Y 279.932,Z 457.083,A -85,B 0,C 180,E1 -17353.967,E2 -17353.967} C_VEL
LIN {X 0,Y 278.116,Z 461.571,A -85,B 0,C 180,E1 -17356.108,E2 -17356.108} C_VEL
LIN {X 0,Y 276.87,Z 465.006,A -85,B 0,C 180,E1 -17358.282,E2 -17358.282} C_VEL
LIN {X 0,Y 276.225,Z 466.776,A -85,B 0,C 180,E1 -17359.739,E2 -17359.739} C_VEL
LIN {X 0,Y 275.775,Z 468.094,A -85,B 0,C 180,E1 -17361.203,E2 -17361.203} C_VEL
LIN {X 0,Y 275.333,Z 469.511,A -85,B 0,C 180,E1 -17364.138,E2 -17364.138} C_VEL
LIN {X 0,Y 275.326,Z 469.616,A -85,B 0,C 180,E1 -17365.606,E2 -17365.606} C_VEL
LIN {X 0,Y 275.356,Z 469.267,A -85,B 0,C 180,E1 -17367.072,E2 -17367.072} C_VEL
LIN {X 0,Y 275.522,Z 468.251,A -85,B 0,C 180,E1 -17368.902,E2 -17368.902} C_VEL
LIN {X 0,Y 275.602,Z 468.812,A -85,B 0,C 180,E1 -17369.998,E2 -17369.998} C_VEL
LIN {X 0,Y 275.405,Z 469.126,A -85,B 0,C 180,E1 -17372.924,E2 -17372.924} C_VEL
LIN {X 0,Y 275.34,Z 468.117,A -85,B 0,C 180,E1 -17375.457,E2 -17375.457} C_VEL
LIN {X 0,Y 275.451,Z 466.58,A -85,B 0,C 180,E1 -17377.328,E2 -17377.328} C_VEL
LIN {X 0,Y 275.897,Z 463.915,A -85,B 0,C 180,E1 -17379.529,E2 -17379.529} C_VEL
LIN {X 0,Y 276.579,Z 460.245,A -85,B 0,C 180,E1 -17381.727,E2 -17381.727} C_VEL
LIN {X 0,Y 277.76,Z 455.468,A -85,B 0,C 180,E1 -17383.907,E2 -17383.907} C_VEL
LIN {X 0,Y 279.337,Z 449.443,A -85,B 0,C 180,E1 -17386.065,E2 -17386.065} C_VEL
LIN {X 0,Y 281.045,Z 442.205,A -85,B 0,C 180,E1 -17388.148,E2 -17388.148} C_VEL
LIN {X 0,Y 283.055,Z 434.36,A -85,B 0,C 180,E1 -17389.96,E2 -17389.96} C_VEL
LIN {X 0,Y 285.583,Z 424.03,A -85,B 0,C 180,E1 -17391.851,E2 -17391.851} C_VEL
LIN {X 0,Y 287.863,Z 413.533,A -85,B 0,C 180,E1 -17393.372,E2 -17393.372} C_VEL
LIN {X 0,Y 289.783,Z 403.411,A -85,B 0,C 180,E1 -17394.538,E2 -17394.538} C_VEL
LIN {X 0,Y 291.829,Z 391.341,A -85,B 0,C 180,E1 -17395.592,E2 -17395.592} C_VEL
LIN {X 0,Y 293.601,Z 377.986,A -85,B 0,C 180,E1 -17396.427,E2 -17396.427} C_VEL
LIN {X 0,Y 294.615,Z 365.514,A -85,B 0,C 180,E1 -17396.95,E2 -17396.95} C_VEL
LIN {X 0,Y 296.587,Z 307.606,A -85,B 0,C 180,E1 -17398.4,E2 -17398.4} C_VEL
LIN {X 0,Y 293.561,Z 284.868,A -85,B 0,C 180,E1 -17399.451,E2 -17399.451} C_VEL
LIN {X 0,Y 290.552,Z 266.549,A -85,B 0,C 180,E1 -17400.402,E2 -17400.402} C_VEL
LIN {X 0,Y 284.893,Z 251.621,A -85,B 0,C 180,E1 -17401.671,E2 -17401.671} C_VEL
LIN {X 0,Y 281.134,Z 242.307,A -85,B 0,C 180,E1 -17402.573,E2 -17402.573} C_VEL
LIN {X 0,Y 278.991,Z 238.729,A -85,B 0,C 180,E1 -17403.082,E2 -17403.082} C_VEL
LIN {X 0,Y 277.487,Z 236.083,A -85,B 0,C 180,E1 -17403.452,E2 -17403.452} C_VEL
LIN {X 0,Y 277.254,Z 234.907,A -85,B 0,C 180,E1 -17403.575,E2 -17403.575} C_VEL
LIN {X 0,Y 277.247,Z 234.949,A -85,B 0,C 180,E1 -17407.47,E2 -17407.47} C_VEL
LIN {X 0,Y 277.171,Z 234.961,A -85,B 0,C 180,E1 -17411.241,E2 -17411.241} C_VEL
LIN {X 0,Y 277.168,Z 234.958,A -85,B 0,C 180,E1 -17415.231,E2 -17415.231} C_VEL
LIN {X 0,Y 277.177,Z 234.939,A -85,B 0,C 180,E1 -17418.758,E2 -17418.758} C_VEL
LIN {X 0,Y 277.247,Z 234.937,A -85,B 0,C 180,E1 -17422.528,E2 -17422.528} C_VEL
LIN {X 0,Y 277.238,Z 234.942,A -85,B 0,C 180,E1 -17426.103,E2 -17426.103} C_VEL
LIN {X 0,Y 277.22,Z 234.928,A -85,B 0,C 180,E1 -17429.534,E2 -17429.534} C_VEL
LIN {X 0,Y 277.245,Z 234.935,A -85,B 0,C 180,E1 -17432.852,E2 -17432.852} C_VEL
LIN {X 0,Y 277.273,Z 234.927,A -85,B 0,C 180,E1 -17436.075,E2 -17436.075} C_VEL
LIN {X 0,Y 277.277,Z 234.936,A -85,B 0,C 180,E1 -17440.762,E2 -17440.762} C_VEL
LIN {X 0,Y 277.4,Z 234.897,A -85,B 0,C 180,E1 -17445.324,E2 -17445.324} C_VEL
LIN {X 0,Y 277.449,Z 234.923,A -85,B 0,C 180,E1 -17449.787,E2 -17449.787} C_VEL
LIN {X 0,Y 277.59,Z 234.889,A -85,B 0,C 180,E1 -17452.728,E2 -17452.728} C_VEL
LIN {X 0,Y 277.799,Z 234.879,A -85,B 0,C 180,E1 -17458.551,E2 -17458.551} C_VEL
LIN {X 0,Y 277.804,Z 234.851,A -85,B 0,C 180,E1 -17461.45,E2 -17461.45} C_VEL
LIN {X 0,Y 277.632,Z 234.895,A -85,B 0,C 180,E1 -17467.272,E2 -17467.272} C_VEL
LIN {X 0,Y 277.453,Z 234.89,A -85,B 0,C 180,E1 -17470.214,E2 -17470.214} C_VEL
LIN {X 0,Y 277.402,Z 234.925,A -85,B 0,C 180,E1 -17474.676,E2 -17474.676} C_VEL
LIN {X 0,Y 277.325,Z 234.93,A -85,B 0,C 180,E1 -17479.236,E2 -17479.236} C_VEL
LIN {X 0,Y 277.313,Z 234.921,A -85,B 0,C 180,E1 -17484.171,E2 -17484.171} C_VEL
LIN {X 0,Y 277.318,Z 234.937,A -85,B 0,C 180,E1 -17487.506,E2 -17487.506} C_VEL
LIN {X 0,Y 277.266,Z 234.939,A -85,B 0,C 180,E1 -17490.483,E2 -17490.483} C_VEL
LIN {X 0,Y 277.241,Z 234.938,A -85,B 0,C 180,E1 -17493.897,E2 -17493.897} C_VEL
LIN {X 0,Y 277.263,Z 234.943,A -85,B 0,C 180,E1 -17497.471,E2 -17497.471} C_VEL
LIN {X 0,Y 277.205,Z 234.951,A -85,B 0,C 180,E1 -17501.238,E2 -17501.238} C_VEL
LIN {X 0,Y 277.202,Z 234.954,A -85,B 0,C 180,E1 -17502.997,E2 -17502.997} C_VEL
LIN {X 0,Y 278.176,Z 237.777,A -85,B 0,C 180,E1 -17503.26,E2 -17503.26} C_VEL
LIN {X 0,Y 279.886,Z 240.161,A -85,B 0,C 180,E1 -17503.611,E2 -17503.611} C_VEL
LIN {X 0,Y 288.783,Z 254.937,A -85,B 0,C 180,E1 -17505.41,E2 -17505.41} C_VEL
LIN {X 0,Y 296.438,Z 269.098,A -85,B 0,C 180,E1 -17506.879,E2 -17506.879} C_VEL
LIN {X 0,Y 298.376,Z 273.131,A -85,B 0,C 180,E1 -17507.248,E2 -17507.248} C_VEL
LIN {X 0,Y 295.752,Z 341.839,A -85,B 0,C 180,E1 -17508.916,E2 -17508.916} C_VEL
LIN {X 0,Y 294.853,Z 355.202,A -85,B 0,C 180,E1 -17509.497,E2 -17509.497} C_VEL
LIN {X 0,Y 293.578,Z 367.471,A -85,B 0,C 180,E1 -17510.31,E2 -17510.31} C_VEL
LIN {X 0,Y 291.751,Z 380.13,A -85,B 0,C 180,E1 -17511.444,E2 -17511.444} C_VEL
LIN {X 0,Y 289.915,Z 390.768,A -85,B 0,C 180,E1 -17512.698,E2 -17512.698} C_VEL
LIN {X 0,Y 287.56,Z 401.593,A -85,B 0,C 180,E1 -17514.304,E2 -17514.304} C_VEL
LIN {X 0,Y 285.515,Z 410.402,A -85,B 0,C 180,E1 -17515.947,E2 -17515.947} C_VEL
LIN {X 0,Y 283.361,Z 418.798,A -85,B 0,C 180,E1 -17517.884,E2 -17517.884} C_VEL
LIN {X 0,Y 281.331,Z 426.152,A -85,B 0,C 180,E1 -17520.027,E2 -17520.027} C_VEL
LIN {X 0,Y 279.561,Z 432.278,A -85,B 0,C 180,E1 -17522.287,E2 -17522.287} C_VEL
LIN {X 0,Y 278.161,Z 437.04,A -85,B 0,C 180,E1 -17524.565,E2 -17524.565} C_VEL
LIN {X 0,Y 277.382,Z 439.523,A -85,B 0,C 180,E1 -17526.086,E2 -17526.086} C_VEL
LIN {X 0,Y 276.718,Z 441.508,A -85,B 0,C 180,E1 -17527.608,E2 -17527.608} C_VEL
LIN {X 0,Y 276.216,Z 443.055,A -85,B 0,C 180,E1 -17529.134,E2 -17529.134} C_VEL
LIN {X 0,Y 275.787,Z 444.116,A -85,B 0,C 180,E1 -17530.655,E2 -17530.655} C_VEL
LIN {X 0,Y 275.494,Z 444.754,A -85,B 0,C 180,E1 -17532.176,E2 -17532.176} C_VEL
LIN {X 0,Y 275.296,Z 444.992,A -85,B 0,C 180,E1 -17533.693,E2 -17533.693} C_VEL
LIN {X 0,Y 275.209,Z 444.502,A -85,B 0,C 180,E1 -17536.028,E2 -17536.028} C_VEL
LIN {X 0,Y 275.232,Z 443.123,A -85,B 0,C 180,E1 -17538.214,E2 -17538.214} C_VEL
LIN {X 0,Y 275.347,Z 441.666,A -85,B 0,C 180,E1 -17539.709,E2 -17539.709} C_VEL
LIN {X 0,Y 275.707,Z 438.642,A -85,B 0,C 180,E1 -17541.942,E2 -17541.942} C_VEL
LIN {X 0,Y 276.146,Z 434.562,A -85,B 0,C 180,E1 -17544.159,E2 -17544.159} C_VEL
LIN {X 0,Y 276.871,Z 428.318,A -85,B 0,C 180,E1 -17546.727,E2 -17546.727} C_VEL
LIN {X 0,Y 277.756,Z 421.516,A -85,B 0,C 180,E1 -17548.914,E2 -17548.914} C_VEL
LIN {X 0,Y 278.981,Z 412.958,A -85,B 0,C 180,E1 -17551.084,E2 -17551.084} C_VEL
LIN {X 0,Y 280.219,Z 404.201,A -85,B 0,C 180,E1 -17552.877,E2 -17552.877} C_VEL
LIN {X 0,Y 281.562,Z 394.592,A -85,B 0,C 180,E1 -17554.475,E2 -17554.475} C_VEL
LIN {X 0,Y 282.916,Z 383.36,A -85,B 0,C 180,E1 -17555.961,E2 -17555.961} C_VEL
LIN {X 0,Y 284.008,Z 372.313,A -85,B 0,C 180,E1 -17557.109,E2 -17557.109} C_VEL
LIN {X 0,Y 284.97,Z 360.263,A -85,B 0,C 180,E1 -17558.065,E2 -17558.065} C_VEL
LIN {X 0,Y 285.698,Z 347.179,A -85,B 0,C 180,E1 -17558.787,E2 -17558.787} C_VEL
LIN {X 0,Y 286.155,Z 333.551,A -85,B 0,C 180,E1 -17559.241,E2 -17559.241} C_VEL
LIN {X 0,Y 287.962,Z 262.431,A -85,B 0,C 180,E1 -17560.981,E2 -17560.981} C_VEL
LIN {X 0,Y 286.979,Z 258.627,A -85,B 0,C 180,E1 -17561.155,E2 -17561.155} C_VEL
LIN {X 0,Y 278.263,Z 237.463,A -85,B 0,C 180,E1 -17562.413,E2 -17562.413} C_VEL
LIN {X 0,Y 277.437,Z 234.928,A -85,B 0,C 180,E1 -17562.599,E2 -17562.599} C_VEL
LIN {X 0,Y 277.412,Z 234.93,A -85,B 0,C 180,E1 -17566.183,E2 -17566.183} C_VEL
LIN {X 0,Y 277.35,Z 234.938,A -85,B 0,C 180,E1 -17570.35,E2 -17570.35} C_VEL
LIN {X 0,Y 277.258,Z 234.95,A -85,B 0,C 180,E1 -17574.14,E2 -17574.14} C_VEL
LIN {X 0,Y 277.242,Z 234.948,A -85,B 0,C 180,E1 -17577.47,E2 -17577.47} C_VEL
LIN {X 0,Y 277.234,Z 234.947,A -85,B 0,C 180,E1 -17580.466,E2 -17580.466} C_VEL
LIN {X 0,Y 277.252,Z 234.95,A -85,B 0,C 180,E1 -17583.897,E2 -17583.897} C_VEL
LIN {X 0,Y 277.257,Z 234.946,A -85,B 0,C 180,E1 -17587.473,E2 -17587.473} C_VEL
LIN {X 0,Y 277.19,Z 234.956,A -85,B 0,C 180,E1 -17591.242,E2 -17591.242} C_VEL
LIN {X 0,Y 277.18,Z 234.956,A -85,B 0,C 180,E1 -17595.233,E2 -17595.233} C_VEL
LIN {X 0,Y 277.183,Z 234.955,A -85,B 0,C 180,E1 -17598.758,E2 -17598.758} C_VEL
LIN {X 0,Y 277.239,Z 234.941,A -85,B 0,C 180,E1 -17602.526,E2 -17602.526} C_VEL
LIN {X 0,Y 277.252,Z 234.946,A -85,B 0,C 180,E1 -17606.104,E2 -17606.104} C_VEL
LIN {X 0,Y 277.235,Z 234.944,A -85,B 0,C 180,E1 -17609.535,E2 -17609.535} C_VEL
LIN {X 0,Y 277.26,Z 234.938,A -85,B 0,C 180,E1 -17612.853,E2 -17612.853} C_VEL
LIN {X 0,Y 277.323,Z 234.933,A -85,B 0,C 180,E1 -17614.906,E2 -17614.906} C_VEL
LIN {X 0,Y 284.101,Z 261.029,A -85,B 0,C 180,E1 -17616.251,E2 -17616.251} C_VEL
LIN {X 0,Y 284.342,Z 264.801,A -85,B 0,C 180,E1 -17616.41,E2 -17616.41} C_VEL
LIN {X 0,Y 283.347,Z 270.55,A -85,B 0,C 180,E1 -17616.603,E2 -17616.603} C_VEL
LIN {X 0,Y 277.007,Z 289.137,A -85,B 0,C 180,E1 -17617.142,E2 -17617.142} C_VEL
LIN {X 0,Y 276.107,Z 294.884,A -85,B 0,C 180,E1 -17617.352,E2 -17617.352} C_VEL
LIN {X 0,Y 274.195,Z 343.886,A -85,B 0,C 180,E1 -17619.363,E2 -17619.363} C_VEL
LIN {X 0,Y 273.649,Z 357.436,A -85,B 0,C 180,E1 -17620.202,E2 -17620.202} C_VEL
LIN {X 0,Y 272.989,Z 369.625,A -85,B 0,C 180,E1 -17621.227,E2 -17621.227} C_VEL
LIN {X 0,Y 272.115,Z 382.054,A -85,B 0,C 180,E1 -17622.572,E2 -17622.572} C_VEL
LIN {X 0,Y 271.175,Z 394.046,A -85,B 0,C 180,E1 -17624.209,E2 -17624.209} C_VEL
LIN {X 0,Y 270.401,Z 405.063,A -85,B 0,C 180,E1 -17626.088,E2 -17626.088} C_VEL
LIN {X 0,Y 269.629,Z 414.05,A -85,B 0,C 180,E1 -17627.964,E2 -17627.964} C_VEL
LIN {X 0,Y 269.057,Z 422.842,A -85,B 0,C 180,E1 -17630.224,E2 -17630.224} C_VEL
LIN {X 0,Y 268.647,Z 429.946,A -85,B 0,C 180,E1 -17632.484,E2 -17632.484} C_VEL
LIN {X 0,Y 268.377,Z 435.86,A -85,B 0,C 180,E1 -17634.872,E2 -17634.872} C_VEL
LIN {X 0,Y 268.373,Z 439.975,A -85,B 0,C 180,E1 -17636.997,E2 -17636.997} C_VEL
LIN {X 0,Y 268.313,Z 442.253,A -85,B 0,C 180,E1 -17638.499,E2 -17638.499} C_VEL
LIN {X 0,Y 268.349,Z 444.088,A -85,B 0,C 180,E1 -17640,E2 -17640} C_VEL
LIN {X 0,Y 268.512,Z 445.499,A -85,B 0,C 180,E1 -17641.499,E2 -17641.499} C_VEL
LIN {X 0,Y 268.785,Z 446.444,A -85,B 0,C 180,E1 -17642.997,E2 -17642.997} C_VEL
LIN {X 0,Y 269.205,Z 446.977,A -85,B 0,C 180,E1 -17644.492,E2 -17644.492} C_VEL
LIN {X 0,Y 269.717,Z 447.111,A -85,B 0,C 180,E1 -17645.982,E2 -17645.982} C_VEL
LIN {X 0,Y 270.131,Z 446.848,A -85,B 0,C 180,E1 -17647.474,E2 -17647.474} C_VEL
LIN {X 0,Y 270.694,Z 446.154,A -85,B 0,C 180,E1 -17648.962,E2 -17648.962} C_VEL
LIN {X 0,Y 271.816,Z 445.008,A -85,B 0,C 180,E1 -17650.427,E2 -17650.427} C_VEL
LIN {X 0,Y 272.924,Z 443.48,A -85,B 0,C 180,E1 -17651.888,E2 -17651.888} C_VEL
LIN {X 0,Y 274.872,Z 440.337,A -85,B 0,C 180,E1 -17654.057,E2 -17654.057} C_VEL
LIN {X 0,Y 277.116,Z 436.179,A -85,B 0,C 180,E1 -17656.199,E2 -17656.199} C_VEL
LIN {X 0,Y 280.275,Z 429.866,A -85,B 0,C 180,E1 -17658.645,E2 -17658.645} C_VEL
LIN {X 0,Y 283.923,Z 421.763,A -85,B 0,C 180,E1 -17661.034,E2 -17661.034} C_VEL
LIN {X 0,Y 287.488,Z 413.071,A -85,B 0,C 180,E1 -17663.025,E2 -17663.025} C_VEL
LIN {X 0,Y 291.458,Z 402.371,A -85,B 0,C 180,E1 -17664.96,E2 -17664.96} C_VEL
LIN {X 0,Y 294.958,Z 391.427,A -85,B 0,C 180,E1 -17666.536,E2 -17666.536} C_VEL
LIN {X 0,Y 298.409,Z 379.286,A -85,B 0,C 180,E1 -17667.91,E2 -17667.91} C_VEL
LIN {X 0,Y 301.613,Z 365.579,A -85,B 0,C 180,E1 -17669.105,E2 -17669.105} C_VEL
LIN {X 0,Y 303.947,Z 353.375,A -85,B 0,C 180,E1 -17669.906,E2 -17669.906} C_VEL
LIN {X 0,Y 306.759,Z 334.455,A -85,B 0,C 180,E1 -17670.794,E2 -17670.794} C_VEL
LIN {X 0,Y 312.257,Z 298.593,A -85,B 0,C 180,E1 -17672.321,E2 -17672.321} C_VEL
LIN {X 0,Y 309.521,Z 293.267,A -85,B 0,C 180,E1 -17673.93,E2 -17673.93} C_VEL
LIN {X 0,Y 307.724,Z 290.064,A -85,B 0,C 180,E1 -17675.139,E2 -17675.139} C_VEL
LIN {X 0,Y 306.062,Z 287.29,A -85,B 0,C 180,E1 -17676.405,E2 -17676.405} C_VEL
LIN {X 0,Y 304.141,Z 284.289,A -85,B 0,C 180,E1 -17678.216,E2 -17678.216} C_VEL
LIN {X 0,Y 301.931,Z 281.618,A -85,B 0,C 180,E1 -17681.372,E2 -17681.372} C_VEL
LIN {X 0,Y 301.249,Z 281.483,A -85,B 0,C 180,E1 -17683.677,E2 -17683.677} C_VEL
LIN {X 0,Y 301.45,Z 282.544,A -85,B 0,C 180,E1 -17686.126,E2 -17686.126} C_VEL
LIN {X 0,Y 302.027,Z 283.998,A -85,B 0,C 180,E1 -17687.619,E2 -17687.619} C_VEL
LIN {X 0,Y 304.559,Z 289.873,A -85,B 0,C 180,E1 -17691.063,E2 -17691.063} C_VEL
LIN {X 0,Y 306.982,Z 296.097,A -85,B 0,C 180,E1 -17693.253,E2 -17693.253} C_VEL
LIN {X 0,Y 308.746,Z 300.871,A -85,B 0,C 180,E1 -17694.576,E2 -17694.576} C_VEL
LIN {X 0,Y 310.064,Z 304.974,A -85,B 0,C 180,E1 -17695.507,E2 -17695.507} C_VEL
LIN {X 0,Y 310.281,Z 315.884,A -85,B 0,C 180,E1 -17696.627,E2 -17696.627} C_VEL
LIN {X 0,Y 302.874,Z 366.262,A -85,B 0,C 180,E1 -17698.817,E2 -17698.817} C_VEL
LIN {X 0,Y 299.959,Z 380.391,A -85,B 0,C 180,E1 -17699.653,E2 -17699.653} C_VEL
LIN {X 0,Y 296.816,Z 392.481,A -85,B 0,C 180,E1 -17700.571,E2 -17700.571} C_VEL
LIN {X 0,Y 292.979,Z 405.701,A -85,B 0,C 180,E1 -17701.914,E2 -17701.914} C_VEL
LIN {X 0,Y 289.019,Z 417.633,A -85,B 0,C 180,E1 -17703.459,E2 -17703.459} C_VEL
LIN {X 0,Y 285.158,Z 428.302,A -85,B 0,C 180,E1 -17705.228,E2 -17705.228} C_VEL
LIN {X 0,Y 281.403,Z 437.964,A -85,B 0,C 180,E1 -17707.224,E2 -17707.224} C_VEL
LIN {X 0,Y 278.114,Z 445.9,A -85,B 0,C 180,E1 -17709.279,E2 -17709.279} C_VEL
LIN {X 0,Y 275.333,Z 452.416,A -85,B 0,C 180,E1 -17711.392,E2 -17711.392} C_VEL
LIN {X 0,Y 273.16,Z 457.713,A -85,B 0,C 180,E1 -17713.558,E2 -17713.558} C_VEL
LIN {X 0,Y 271.241,Z 461.95,A -85,B 0,C 180,E1 -17715.749,E2 -17715.749} C_VEL
LIN {X 0,Y 269.904,Z 465.177,A -85,B 0,C 180,E1 -17717.975,E2 -17717.975} C_VEL
LIN {X 0,Y 268.733,Z 467.972,A -85,B 0,C 180,E1 -17720.971,E2 -17720.971} C_VEL
LIN {X 0,Y 268.387,Z 468.777,A -85,B 0,C 180,E1 -17722.475,E2 -17722.475} C_VEL
LIN {X 0,Y 268.215,Z 469.182,A -85,B 0,C 180,E1 -17724.69,E2 -17724.69} C_VEL
LIN {X 0,Y 268.286,Z 468.655,A -85,B 0,C 180,E1 -17726.995,E2 -17726.995} C_VEL
LIN {X 0,Y 268.411,Z 467.749,A -85,B 0,C 180,E1 -17728.686,E2 -17728.686} C_VEL
LIN {X 0,Y 268.509,Z 468.453,A -85,B 0,C 180,E1 -17729.998,E2 -17729.998} C_VEL
LIN {X 0,Y 268.328,Z 468.825,A -85,B 0,C 180,E1 -17733.001,E2 -17733.001} C_VEL
LIN {X 0,Y 268.248,Z 467.621,A -85,B 0,C 180,E1 -17736.014,E2 -17736.014} C_VEL
LIN {X 0,Y 268.675,Z 464.742,A -85,B 0,C 180,E1 -17739.028,E2 -17739.028} C_VEL
LIN {X 0,Y 269.313,Z 461.469,A -85,B 0,C 180,E1 -17741.285,E2 -17741.285} C_VEL
LIN {X 0,Y 270.352,Z 457.14,A -85,B 0,C 180,E1 -17743.529,E2 -17743.529} C_VEL
LIN {X 0,Y 272.247,Z 450.607,A -85,B 0,C 180,E1 -17746.11,E2 -17746.11} C_VEL
LIN {X 0,Y 274.175,Z 442.824,A -85,B 0,C 180,E1 -17748.481,E2 -17748.481} C_VEL
LIN {X 0,Y 276.397,Z 434.594,A -85,B 0,C 180,E1 -17750.462,E2 -17750.462} C_VEL
LIN {X 0,Y 278.798,Z 425.486,A -85,B 0,C 180,E1 -17752.216,E2 -17752.216} C_VEL
LIN {X 0,Y 281.157,Z 415.358,A -85,B 0,C 180,E1 -17753.768,E2 -17753.768} C_VEL
LIN {X 0,Y 283.381,Z 404.163,A -85,B 0,C 180,E1 -17755.13,E2 -17755.13} C_VEL
LIN {X 0,Y 285.486,Z 392.525,A -85,B 0,C 180,E1 -17756.203,E2 -17756.203} C_VEL
LIN {X 0,Y 287.314,Z 379.709,A -85,B 0,C 180,E1 -17757.052,E2 -17757.052} C_VEL
LIN {X 0,Y 288.542,Z 366.219,A -85,B 0,C 180,E1 -17757.661,E2 -17757.661} C_VEL
LIN {X 0,Y 290.656,Z 308.607,A -85,B 0,C 180,E1 -17759.133,E2 -17759.133} C_VEL
LIN {X 0,Y 287.739,Z 286.308,A -85,B 0,C 180,E1 -17760.197,E2 -17760.197} C_VEL
LIN {X 0,Y 284.976,Z 269.176,A -85,B 0,C 180,E1 -17761.115,E2 -17761.115} C_VEL
LIN {X 0,Y 279.207,Z 253.929,A -85,B 0,C 180,E1 -17762.465,E2 -17762.465} C_VEL
LIN {X 0,Y 275.956,Z 246.17,A -85,B 0,C 180,E1 -17763.24,E2 -17763.24} C_VEL
LIN {X 0,Y 274.028,Z 243.073,A -85,B 0,C 180,E1 -17763.683,E2 -17763.683} C_VEL
LIN {X 0,Y 271.935,Z 239.635,A -85,B 0,C 180,E1 -17764.206,E2 -17764.206} C_VEL
LIN {X 0,Y 270.432,Z 236.978,A -85,B 0,C 180,E1 -17764.598,E2 -17764.598} C_VEL
LIN {X 0,Y 270.183,Z 235.793,A -85,B 0,C 180,E1 -17764.735,E2 -17764.735} C_VEL
LIN {X 0,Y 270.162,Z 235.82,A -85,B 0,C 180,E1 -17768.701,E2 -17768.701} C_VEL
LIN {X 0,Y 270.142,Z 235.82,A -85,B 0,C 180,E1 -17773.244,E2 -17773.244} C_VEL
LIN {X 0,Y 270.144,Z 235.819,A -85,B 0,C 180,E1 -17777.437,E2 -17777.437} C_VEL
LIN {X 0,Y 270.2,Z 235.827,A -85,B 0,C 180,E1 -17781.373,E2 -17781.373} C_VEL
LIN {X 0,Y 270.19,Z 235.805,A -85,B 0,C 180,E1 -17785.093,E2 -17785.093} C_VEL
LIN {X 0,Y 270.163,Z 235.811,A -85,B 0,C 180,E1 -17789.14,E2 -17789.14} C_VEL
LIN {X 0,Y 270.18,Z 235.807,A -85,B 0,C 180,E1 -17792.176,E2 -17792.176} C_VEL
LIN {X 0,Y 270.219,Z 235.813,A -85,B 0,C 180,E1 -17795.542,E2 -17795.542} C_VEL
LIN {X 0,Y 270.215,Z 235.812,A -85,B 0,C 180,E1 -17800.238,E2 -17800.238} C_VEL
LIN {X 0,Y 270.359,Z 235.777,A -85,B 0,C 180,E1 -17804.933,E2 -17804.933} C_VEL
LIN {X 0,Y 270.401,Z 235.801,A -85,B 0,C 180,E1 -17809.518,E2 -17809.518} C_VEL
LIN {X 0,Y 270.552,Z 235.767,A -85,B 0,C 180,E1 -17812.538,E2 -17812.538} C_VEL
LIN {X 0,Y 270.765,Z 235.755,A -85,B 0,C 180,E1 -17818.513,E2 -17818.513} C_VEL
LIN {X 0,Y 270.769,Z 235.726,A -85,B 0,C 180,E1 -17821.488,E2 -17821.488} C_VEL
LIN {X 0,Y 270.59,Z 235.773,A -85,B 0,C 180,E1 -17827.462,E2 -17827.462} C_VEL
LIN {X 0,Y 270.405,Z 235.767,A -85,B 0,C 180,E1 -17830.483,E2 -17830.483} C_VEL
LIN {X 0,Y 270.37,Z 235.8,A -85,B 0,C 180,E1 -17835.067,E2 -17835.067} C_VEL
LIN {X 0,Y 270.289,Z 235.81,A -85,B 0,C 180,E1 -17839.757,E2 -17839.757} C_VEL
LIN {X 0,Y 270.268,Z 235.801,A -85,B 0,C 180,E1 -17844.587,E2 -17844.587} C_VEL
LIN {X 0,Y 270.264,Z 235.813,A -85,B 0,C 180,E1 -17847.91,E2 -17847.91} C_VEL
LIN {X 0,Y 270.178,Z 235.83,A -85,B 0,C 180,E1 -17851.35,E2 -17851.35} C_VEL
LIN {X 0,Y 270.197,Z 235.819,A -85,B 0,C 180,E1 -17854.907,E2 -17854.907} C_VEL
LIN {X 0,Y 270.193,Z 235.821,A -85,B 0,C 180,E1 -17858.712,E2 -17858.712} C_VEL
LIN {X 0,Y 270.142,Z 235.828,A -85,B 0,C 180,E1 -17861.836,E2 -17861.836} C_VEL
LIN {X 0,Y 271.139,Z 238.68,A -85,B 0,C 180,E1 -17862.112,E2 -17862.112} C_VEL
LIN {X 0,Y 272.939,Z 241.095,A -85,B 0,C 180,E1 -17862.503,E2 -17862.503} C_VEL
LIN {X 0,Y 281.908,Z 255.719,A -85,B 0,C 180,E1 -17864.42,E2 -17864.42} C_VEL
LIN {X 0,Y 289.778,Z 270.067,A -85,B 0,C 180,E1 -17866.007,E2 -17866.007} C_VEL
LIN {X 0,Y 292.386,Z 275.307,A -85,B 0,C 180,E1 -17866.52,E2 -17866.52} C_VEL
LIN {X 0,Y 289.772,Z 342.009,A -85,B 0,C 180,E1 -17868.171,E2 -17868.171} C_VEL
LIN {X 0,Y 288.851,Z 355.416,A -85,B 0,C 180,E1 -17868.763,E2 -17868.763} C_VEL
LIN {X 0,Y 287.488,Z 367.724,A -85,B 0,C 180,E1 -17869.587,E2 -17869.587} C_VEL
LIN {X 0,Y 285.673,Z 379.927,A -85,B 0,C 180,E1 -17870.694,E2 -17870.694} C_VEL
LIN {X 0,Y 283.586,Z 391.476,A -85,B 0,C 180,E1 -17872.078,E2 -17872.078} C_VEL
LIN {X 0,Y 281.04,Z 402.667,A -85,B 0,C 180,E1 -17873.789,E2 -17873.789} C_VEL
LIN {X 0,Y 278.916,Z 411.345,A -85,B 0,C 180,E1 -17875.465,E2 -17875.465} C_VEL
LIN {X 0,Y 276.898,Z 418.784,A -85,B 0,C 180,E1 -17877.225,E2 -17877.225} C_VEL
LIN {X 0,Y 274.546,Z 426.86,A -85,B 0,C 180,E1 -17879.633,E2 -17879.633} C_VEL
LIN {X 0,Y 272.919,Z 432.134,A -85,B 0,C 180,E1 -17881.616,E2 -17881.616} C_VEL
LIN {X 0,Y 271.43,Z 436.886,A -85,B 0,C 180,E1 -17883.887,E2 -17883.887} C_VEL
LIN {X 0,Y 270.226,Z 440.561,A -85,B 0,C 180,E1 -17886.228,E2 -17886.228} C_VEL
LIN {X 0,Y 269.309,Z 443.137,A -85,B 0,C 180,E1 -17888.573,E2 -17888.573} C_VEL
LIN {X 0,Y 268.805,Z 444.369,A -85,B 0,C 180,E1 -17890.262,E2 -17890.262} C_VEL
LIN {X 0,Y 268.254,Z 445.287,A -85,B 0,C 180,E1 -17893.252,E2 -17893.252} C_VEL
LIN {X 0,Y 268.134,Z 444.824,A -85,B 0,C 180,E1 -17895.886,E2 -17895.886} C_VEL
LIN {X 0,Y 268.14,Z 443.624,A -85,B 0,C 180,E1 -17897.898,E2 -17897.898} C_VEL
LIN {X 0,Y 268.216,Z 442.252,A -85,B 0,C 180,E1 -17899.433,E2 -17899.433} C_VEL
LIN {X 0,Y 268.558,Z 439.338,A -85,B 0,C 180,E1 -17901.726,E2 -17901.726} C_VEL
LIN {X 0,Y 269.026,Z 435.382,A -85,B 0,C 180,E1 -17904.004,E2 -17904.004} C_VEL
LIN {X 0,Y 269.617,Z 430.272,A -85,B 0,C 180,E1 -17906.265,E2 -17906.265} C_VEL
LIN {X 0,Y 270.46,Z 423.829,A -85,B 0,C 180,E1 -17908.513,E2 -17908.513} C_VEL
LIN {X 0,Y 271.648,Z 415.807,A -85,B 0,C 180,E1 -17910.743,E2 -17910.743} C_VEL
LIN {X 0,Y 272.882,Z 407.605,A -85,B 0,C 180,E1 -17912.585,E2 -17912.585} C_VEL
LIN {X 0,Y 274.331,Z 397.515,A -85,B 0,C 180,E1 -17914.409,E2 -17914.409} C_VEL
LIN {X 0,Y 275.662,Z 387.565,A -85,B 0,C 180,E1 -17915.855,E2 -17915.855} C_VEL
LIN {X 0,Y 276.898,Z 376.474,A -85,B 0,C 180,E1 -17917.142,E2 -17917.142} C_VEL
LIN {X 0,Y 277.809,Z 364.954,A -85,B 0,C 180,E1 -17918.183,E2 -17918.183} C_VEL
LIN {X 0,Y 278.733,Z 351.855,A -85,B 0,C 180,E1 -17919.023,E2 -17919.023} C_VEL
LIN {X 0,Y 279.281,Z 339.211,A -85,B 0,C 180,E1 -17919.553,E2 -17919.553} C_VEL
LIN {X 0,Y 281.271,Z 263.103,A -85,B 0,C 180,E1 -17921.472,E2 -17921.472} C_VEL
LIN {X 0,Y 275.404,Z 248.004,A -85,B 0,C 180,E1 -17922.357,E2 -17922.357} C_VEL
LIN {X 0,Y 270.494,Z 236.377,A -85,B 0,C 180,E1 -17923.101,E2 -17923.101} C_VEL
LIN {X 0,Y 270.378,Z 235.805,A -85,B 0,C 180,E1 -17923.149,E2 -17923.149} C_VEL
LIN {X 0,Y 270.36,Z 235.809,A -85,B 0,C 180,E1 -17926.617,E2 -17926.617} C_VEL
LIN {X 0,Y 270.297,Z 235.816,A -85,B 0,C 180,E1 -17930.602,E2 -17930.602} C_VEL
LIN {X 0,Y 270.19,Z 235.829,A -85,B 0,C 180,E1 -17934.595,E2 -17934.595} C_VEL
LIN {X 0,Y 270.19,Z 235.83,A -85,B 0,C 180,E1 -17937.919,E2 -17937.919} C_VEL
LIN {X 0,Y 270.175,Z 235.826,A -85,B 0,C 180,E1 -17941.351,E2 -17941.351} C_VEL
LIN {X 0,Y 270.204,Z 235.824,A -85,B 0,C 180,E1 -17944.907,E2 -17944.907} C_VEL
LIN {X 0,Y 270.204,Z 235.825,A -85,B 0,C 180,E1 -17948.711,E2 -17948.711} C_VEL
LIN {X 0,Y 270.154,Z 235.827,A -85,B 0,C 180,E1 -17953.245,E2 -17953.245} C_VEL
LIN {X 0,Y 270.157,Z 235.833,A -85,B 0,C 180,E1 -17957.438,E2 -17957.438} C_VEL
LIN {X 0,Y 270.159,Z 235.823,A -85,B 0,C 180,E1 -17961.365,E2 -17961.365} C_VEL
LIN {X 0,Y 270.204,Z 235.827,A -85,B 0,C 180,E1 -17965.094,E2 -17965.094} C_VEL
LIN {X 0,Y 270.178,Z 235.825,A -85,B 0,C 180,E1 -17969.142,E2 -17969.142} C_VEL
LIN {X 0,Y 270.22,Z 235.814,A -85,B 0,C 180,E1 -17973.759,E2 -17973.759} C_VEL
LIN {X 0,Y 270.299,Z 235.975,A -85,B 0,C 180,E1 -17974.673,E2 -17974.673} C_VEL
LIN {X 0,Y 277.302,Z 263.005,A -85,B 0,C 180,E1 -17976.077,E2 -17976.077} C_VEL
LIN {X 0,Y 276.107,Z 294.884,A -85,B 0,C 180,E1 -17977.352,E2 -17977.352} C_VEL
LIN {X 0,Y 275.181,Z 300.631,A -85,B 0,C 180,E1 -17977.562,E2 -17977.562} C_VEL
LIN {X 0,Y 268.815,Z 319.181,A -85,B 0,C 180,E1 -17978.169,E2 -17978.169} C_VEL
LIN {X 0,Y 267.931,Z 324.926,A -85,B 0,C 180,E1 -17978.393,E2 -17978.393} C_VEL
LIN {X 0,Y 267.078,Z 346.952,A -85,B 0,C 180,E1 -17979.393,E2 -17979.393} C_VEL
LIN {X 0,Y 266.402,Z 360.732,A -85,B 0,C 180,E1 -17980.344,E2 -17980.344} C_VEL
LIN {X 0,Y 265.615,Z 373.115,A -85,B 0,C 180,E1 -17981.487,E2 -17981.487} C_VEL
LIN {X 0,Y 264.866,Z 384.314,A -85,B 0,C 180,E1 -17982.796,E2 -17982.796} C_VEL
LIN {X 0,Y 263.944,Z 396.368,A -85,B 0,C 180,E1 -17984.557,E2 -17984.557} C_VEL
LIN {X 0,Y 263.132,Z 407.01,A -85,B 0,C 180,E1 -17986.484,E2 -17986.484} C_VEL
LIN {X 0,Y 262.355,Z 417.269,A -85,B 0,C 180,E1 -17988.801,E2 -17988.801} C_VEL
LIN {X 0,Y 261.808,Z 425.496,A -85,B 0,C 180,E1 -17991.12,E2 -17991.12} C_VEL
LIN {X 0,Y 261.523,Z 431.128,A -85,B 0,C 180,E1 -17993.054,E2 -17993.054} C_VEL
LIN {X 0,Y 261.276,Z 436.574,A -85,B 0,C 180,E1 -17995.371,E2 -17995.371} C_VEL
LIN {X 0,Y 261.268,Z 440.812,A -85,B 0,C 180,E1 -17997.687,E2 -17997.687} C_VEL
LIN {X 0,Y 261.269,Z 443.956,A -85,B 0,C 180,E1 -18000,E2 -18000} C_VEL
LIN {X 0,Y 261.432,Z 445.483,A -85,B 0,C 180,E1 -18001.54,E2 -18001.54} C_VEL
LIN {X 0,Y 261.713,Z 446.607,A -85,B 0,C 180,E1 -18003.078,E2 -18003.078} C_VEL
LIN {X 0,Y 262.146,Z 447.29,A -85,B 0,C 180,E1 -18004.613,E2 -18004.613} C_VEL
LIN {X 0,Y 262.67,Z 447.541,A -85,B 0,C 180,E1 -18006.143,E2 -18006.143} C_VEL
LIN {X 0,Y 263.742,Z 446.897,A -85,B 0,C 180,E1 -18009.2,E2 -18009.2} C_VEL
LIN {X 0,Y 264.907,Z 445.925,A -85,B 0,C 180,E1 -18010.702,E2 -18010.702} C_VEL
LIN {X 0,Y 267.37,Z 442.727,A -85,B 0,C 180,E1 -18013.684,E2 -18013.684} C_VEL
LIN {X 0,Y 269.651,Z 439.187,A -85,B 0,C 180,E1 -18015.882,E2 -18015.882} C_VEL
LIN {X 0,Y 272.323,Z 434.577,A -85,B 0,C 180,E1 -18018.04,E2 -18018.04} C_VEL
LIN {X 0,Y 275.372,Z 428.812,A -85,B 0,C 180,E1 -18020.154,E2 -18020.154} C_VEL
LIN {X 0,Y 278.834,Z 421.701,A -85,B 0,C 180,E1 -18022.214,E2 -18022.214} C_VEL
LIN {X 0,Y 282.687,Z 412.93,A -85,B 0,C 180,E1 -18024.218,E2 -18024.218} C_VEL
LIN {X 0,Y 286.939,Z 402.176,A -85,B 0,C 180,E1 -18026.159,E2 -18026.159} C_VEL
LIN {X 0,Y 291.098,Z 389.956,A -85,B 0,C 180,E1 -18027.89,E2 -18027.89} C_VEL
LIN {X 0,Y 294.386,Z 378.94,A -85,B 0,C 180,E1 -18029.105,E2 -18029.105} C_VEL
LIN {X 0,Y 297.773,Z 365.283,A -85,B 0,C 180,E1 -18030.297,E2 -18030.297} C_VEL
LIN {X 0,Y 300.406,Z 352.206,A -85,B 0,C 180,E1 -18031.123,E2 -18031.123} C_VEL
LIN {X 0,Y 303.964,Z 329.684,A -85,B 0,C 180,E1 -18032.169,E2 -18032.169} C_VEL
LIN {X 0,Y 308.434,Z 302.687,A -85,B 0,C 180,E1 -18033.315,E2 -18033.315} C_VEL
LIN {X 0,Y 305.881,Z 297.446,A -85,B 0,C 180,E1 -18035.058,E2 -18035.058} C_VEL
LIN {X 0,Y 303.888,Z 293.918,A -85,B 0,C 180,E1 -18036.649,E2 -18036.649} C_VEL
LIN {X 0,Y 301.96,Z 290.818,A -85,B 0,C 180,E1 -18038.595,E2 -18038.595} C_VEL
LIN {X 0,Y 300.102,Z 288.468,A -85,B 0,C 180,E1 -18041.46,E2 -18041.46} C_VEL
LIN {X 0,Y 299.427,Z 288.428,A -85,B 0,C 180,E1 -18044.011,E2 -18044.011} C_VEL
LIN {X 0,Y 299.749,Z 289.674,A -85,B 0,C 180,E1 -18046.415,E2 -18046.415} C_VEL
LIN {X 0,Y 300.191,Z 291.167,A -85,B 0,C 180,E1 -18047.666,E2 -18047.666} C_VEL
LIN {X 0,Y 302.333,Z 296.525,A -85,B 0,C 180,E1 -18050.761,E2 -18050.761} C_VEL
LIN {X 0,Y 304.378,Z 302.302,A -85,B 0,C 180,E1 -18052.812,E2 -18052.812} C_VEL
LIN {X 0,Y 306.155,Z 307.63,A -85,B 0,C 180,E1 -18054.274,E2 -18054.274} C_VEL
LIN {X 0,Y 306.613,Z 309.598,A -85,B 0,C 180,E1 -18054.685,E2 -18054.685} C_VEL
LIN {X 0,Y 306.553,Z 318.157,A -85,B 0,C 180,E1 -18055.564,E2 -18055.564} C_VEL
LIN {X 0,Y 298.997,Z 365.936,A -85,B 0,C 180,E1 -18057.672,E2 -18057.672} C_VEL
LIN {X 0,Y 295.906,Z 379.846,A -85,B 0,C 180,E1 -18058.497,E2 -18058.497} C_VEL
LIN {X 0,Y 292.377,Z 392.68,A -85,B 0,C 180,E1 -18059.482,E2 -18059.482} C_VEL
LIN {X 0,Y 288.34,Z 405.616,A -85,B 0,C 180,E1 -18060.823,E2 -18060.823} C_VEL
LIN {X 0,Y 284.117,Z 417.397,A -85,B 0,C 180,E1 -18062.365,E2 -18062.365} C_VEL
LIN {X 0,Y 280.378,Z 427.084,A -85,B 0,C 180,E1 -18063.98,E2 -18063.98} C_VEL
LIN {X 0,Y 276.306,Z 436.798,A -85,B 0,C 180,E1 -18065.984,E2 -18065.984} C_VEL
LIN {X 0,Y 272.599,Z 445.126,A -85,B 0,C 180,E1 -18068.145,E2 -18068.145} C_VEL
LIN {X 0,Y 269.577,Z 451.437,A -85,B 0,C 180,E1 -18070.187,E2 -18070.187} C_VEL
LIN {X 0,Y 267.15,Z 456.803,A -85,B 0,C 180,E1 -18072.388,E2 -18072.388} C_VEL
LIN {X 0,Y 264.966,Z 461.13,A -85,B 0,C 180,E1 -18074.617,E2 -18074.617} C_VEL
LIN {X 0,Y 263.798,Z 463.419,A -85,B 0,C 180,E1 -18076.125,E2 -18076.125} C_VEL
LIN {X 0,Y 262.236,Z 466.777,A -85,B 0,C 180,E1 -18079.185,E2 -18079.185} C_VEL
LIN {X 0,Y 261.711,Z 467.855,A -85,B 0,C 180,E1 -18080.726,E2 -18080.726} C_VEL
LIN {X 0,Y 261.178,Z 468.741,A -85,B 0,C 180,E1 -18083.819,E2 -18083.819} C_VEL
LIN {X 0,Y 261.173,Z 468.589,A -85,B 0,C 180,E1 -18085.368,E2 -18085.368} C_VEL
LIN {X 0,Y 261.279,Z 467.302,A -85,B 0,C 180,E1 -18088.071,E2 -18088.071} C_VEL
LIN {X 0,Y 261.288,Z 467.206,A -85,B 0,C 180,E1 -18088.457,E2 -18088.457} C_VEL
LIN {X 0,Y 261.419,Z 468.082,A -85,B 0,C 180,E1 -18089.998,E2 -18089.998} C_VEL
LIN {X 0,Y 261.279,Z 468.507,A -85,B 0,C 180,E1 -18091.54,E2 -18091.54} C_VEL
LIN {X 0,Y 261.229,Z 468.522,A -85,B 0,C 180,E1 -18093.083,E2 -18093.083} C_VEL
LIN {X 0,Y 261.161,Z 467.382,A -85,B 0,C 180,E1 -18096.178,E2 -18096.178} C_VEL
LIN {X 0,Y 261.315,Z 466.184,A -85,B 0,C 180,E1 -18097.726,E2 -18097.726} C_VEL
LIN {X 0,Y 261.823,Z 463.63,A -85,B 0,C 180,E1 -18100.046,E2 -18100.046} C_VEL
LIN {X 0,Y 262.605,Z 460.082,A -85,B 0,C 180,E1 -18102.361,E2 -18102.361} C_VEL
LIN {X 0,Y 263.963,Z 455.438,A -85,B 0,C 180,E1 -18104.65,E2 -18104.65} C_VEL
LIN {X 0,Y 265.65,Z 449.559,A -85,B 0,C 180,E1 -18106.917,E2 -18106.917} C_VEL
LIN {X 0,Y 267.837,Z 441.506,A -85,B 0,C 180,E1 -18109.367,E2 -18109.367} C_VEL
LIN {X 0,Y 270.255,Z 433.199,A -85,B 0,C 180,E1 -18111.349,E2 -18111.349} C_VEL
LIN {X 0,Y 273.046,Z 422.734,A -85,B 0,C 180,E1 -18113.31,E2 -18113.31} C_VEL
LIN {X 0,Y 275.56,Z 412.102,A -85,B 0,C 180,E1 -18114.885,E2 -18114.885} C_VEL
LIN {X 0,Y 277.689,Z 401.759,A -85,B 0,C 180,E1 -18116.086,E2 -18116.086} C_VEL
LIN {X 0,Y 279.861,Z 389.356,A -85,B 0,C 180,E1 -18117.175,E2 -18117.175} C_VEL
LIN {X 0,Y 281.659,Z 376.28,A -85,B 0,C 180,E1 -18117.994,E2 -18117.994} C_VEL
LIN {X 0,Y 282.723,Z 363.469,A -85,B 0,C 180,E1 -18118.516,E2 -18118.516} C_VEL
LIN {X 0,Y 284.743,Z 309.244,A -85,B 0,C 180,E1 -18119.917,E2 -18119.917} C_VEL
LIN {X 0,Y 281.79,Z 286.813,A -85,B 0,C 180,E1 -18121.034,E2 -18121.034} C_VEL
LIN {X 0,Y 279.416,Z 271.741,A -85,B 0,C 180,E1 -18121.864,E2 -18121.864} C_VEL
LIN {X 0,Y 272.536,Z 253.428,A -85,B 0,C 180,E1 -18123.565,E2 -18123.565} C_VEL
LIN {X 0,Y 270.472,Z 249.124,A -85,B 0,C 180,E1 -18124.061,E2 -18124.061} C_VEL
LIN {X 0,Y 265.772,Z 241.697,A -85,B 0,C 180,E1 -18125.187,E2 -18125.187} C_VEL
LIN {X 0,Y 263.513,Z 238.222,A -85,B 0,C 180,E1 -18125.791,E2 -18125.791} C_VEL
LIN {X 0,Y 263.153,Z 236.69,A -85,B 0,C 180,E1 -18125.981,E2 -18125.981} C_VEL
LIN {X 0,Y 263.067,Z 236.706,A -85,B 0,C 180,E1 -18129.877,E2 -18129.877} C_VEL
LIN {X 0,Y 263.07,Z 236.702,A -85,B 0,C 180,E1 -18133.993,E2 -18133.993} C_VEL
LIN {X 0,Y 263.073,Z 236.694,A -85,B 0,C 180,E1 -18138.416,E2 -18138.416} C_VEL
LIN {X 0,Y 263.149,Z 236.7,A -85,B 0,C 180,E1 -18142.102,E2 -18142.102} C_VEL
LIN {X 0,Y 263.144,Z 236.692,A -85,B 0,C 180,E1 -18145.885,E2 -18145.885} C_VEL
LIN {X 0,Y 263.101,Z 236.685,A -85,B 0,C 180,E1 -18149.501,E2 -18149.501} C_VEL
LIN {X 0,Y 263.108,Z 236.697,A -85,B 0,C 180,E1 -18152.994,E2 -18152.994} C_VEL
LIN {X 0,Y 263.135,Z 236.681,A -85,B 0,C 180,E1 -18156.383,E2 -18156.383} C_VEL
LIN {X 0,Y 263.2,Z 236.674,A -85,B 0,C 180,E1 -18159.689,E2 -18159.689} C_VEL
LIN {X 0,Y 263.301,Z 236.66,A -85,B 0,C 180,E1 -18164.519,E2 -18164.519} C_VEL
LIN {X 0,Y 263.341,Z 236.678,A -85,B 0,C 180,E1 -18169.233,E2 -18169.233} C_VEL
LIN {X 0,Y 263.516,Z 236.645,A -85,B 0,C 180,E1 -18172.337,E2 -18172.337} C_VEL
LIN {X 0,Y 263.729,Z 236.632,A -85,B 0,C 180,E1 -18178.473,E2 -18178.473} C_VEL
LIN {X 0,Y 263.732,Z 236.601,A -85,B 0,C 180,E1 -18181.527,E2 -18181.527} C_VEL
LIN {X 0,Y 263.55,Z 236.646,A -85,B 0,C 180,E1 -18187.663,E2 -18187.663} C_VEL
LIN {X 0,Y 263.347,Z 236.646,A -85,B 0,C 180,E1 -18190.767,E2 -18190.767} C_VEL
LIN {X 0,Y 263.316,Z 236.672,A -85,B 0,C 180,E1 -18195.481,E2 -18195.481} C_VEL
LIN {X 0,Y 263.255,Z 236.693,A -85,B 0,C 180,E1 -18200.308,E2 -18200.308} C_VEL
LIN {X 0,Y 263.202,Z 236.689,A -85,B 0,C 180,E1 -18205.292,E2 -18205.292} C_VEL
LIN {X 0,Y 263.16,Z 236.689,A -85,B 0,C 180,E1 -18208.733,E2 -18208.733} C_VEL
LIN {X 0,Y 263.127,Z 236.71,A -85,B 0,C 180,E1 -18212.29,E2 -18212.29} C_VEL
LIN {X 0,Y 263.186,Z 236.704,A -85,B 0,C 180,E1 -18216.767,E2 -18216.767} C_VEL
LIN {X 0,Y 263.151,Z 236.709,A -85,B 0,C 180,E1 -18220.585,E2 -18220.585} C_VEL
LIN {X 0,Y 264.178,Z 239.631,A -85,B 0,C 180,E1 -18220.896,E2 -18220.896} C_VEL
LIN {X 0,Y 265.933,Z 241.939,A -85,B 0,C 180,E1 -18221.301,E2 -18221.301} C_VEL
LIN {X 0,Y 275.673,Z 257.546,A -85,B 0,C 180,E1 -18223.499,E2 -18223.499} C_VEL
LIN {X 0,Y 284.165,Z 272.916,A -85,B 0,C 180,E1 -18225.294,E2 -18225.294} C_VEL
LIN {X 0,Y 286.514,Z 277.676,A -85,B 0,C 180,E1 -18225.778,E2 -18225.778} C_VEL
LIN {X 0,Y 283.854,Z 341.703,A -85,B 0,C 180,E1 -18227.377,E2 -18227.377} C_VEL
LIN {X 0,Y 282.891,Z 355.462,A -85,B 0,C 180,E1 -18227.985,E2 -18227.985} C_VEL
LIN {X 0,Y 281.608,Z 366.764,A -85,B 0,C 180,E1 -18228.732,E2 -18228.732} C_VEL
LIN {X 0,Y 279.649,Z 379.742,A -85,B 0,C 180,E1 -18229.912,E2 -18229.912} C_VEL
LIN {X 0,Y 277.636,Z 390.475,A -85,B 0,C 180,E1 -18231.187,E2 -18231.187} C_VEL
LIN {X 0,Y 275.343,Z 400.509,A -85,B 0,C 180,E1 -18232.686,E2 -18232.686} C_VEL
LIN {X 0,Y 272.785,Z 410.499,A -85,B 0,C 180,E1 -18234.574,E2 -18234.574} C_VEL
LIN {X 0,Y 270.389,Z 419.035,A -85,B 0,C 180,E1 -18236.599,E2 -18236.599} C_VEL
LIN {X 0,Y 268.115,Z 426.443,A -85,B 0,C 180,E1 -18238.824,E2 -18238.824} C_VEL
LIN {X 0,Y 266.265,Z 432.18,A -85,B 0,C 180,E1 -18240.993,E2 -18240.993} C_VEL
LIN {X 0,Y 264.747,Z 436.734,A -85,B 0,C 180,E1 -18243.176,E2 -18243.176} C_VEL
LIN {X 0,Y 263.738,Z 439.693,A -85,B 0,C 180,E1 -18244.962,E2 -18244.962} C_VEL
LIN {X 0,Y 263.054,Z 441.558,A -85,B 0,C 180,E1 -18246.377,E2 -18246.377} C_VEL
LIN {X 0,Y 262.425,Z 443.218,A -85,B 0,C 180,E1 -18247.982,E2 -18247.982} C_VEL
LIN {X 0,Y 261.786,Z 444.693,A -85,B 0,C 180,E1 -18249.99,E2 -18249.99} C_VEL
LIN {X 0,Y 261.213,Z 445.583,A -85,B 0,C 180,E1 -18252.787,E2 -18252.787} C_VEL
LIN {X 0,Y 261.042,Z 445.141,A -85,B 0,C 180,E1 -18255.751,E2 -18255.751} C_VEL
LIN {X 0,Y 261.039,Z 444.127,A -85,B 0,C 180,E1 -18257.564,E2 -18257.564} C_VEL
LIN {X 0,Y 261.091,Z 442.807,A -85,B 0,C 180,E1 -18259.141,E2 -18259.141} C_VEL
LIN {X 0,Y 261.418,Z 440,A -85,B 0,C 180,E1 -18261.499,E2 -18261.499} C_VEL
LIN {X 0,Y 261.894,Z 436.157,A -85,B 0,C 180,E1 -18263.84,E2 -18263.84} C_VEL
LIN {X 0,Y 262.494,Z 431.189,A -85,B 0,C 180,E1 -18266.164,E2 -18266.164} C_VEL
LIN {X 0,Y 263.35,Z 424.922,A -85,B 0,C 180,E1 -18268.472,E2 -18268.472} C_VEL
LIN {X 0,Y 264.542,Z 417.061,A -85,B 0,C 180,E1 -18270.763,E2 -18270.763} C_VEL
LIN {X 0,Y 265.768,Z 409.046,A -85,B 0,C 180,E1 -18272.654,E2 -18272.654} C_VEL
LIN {X 0,Y 267.245,Z 399.283,A -85,B 0,C 180,E1 -18274.527,E2 -18274.527} C_VEL
LIN {X 0,Y 268.79,Z 388.106,A -85,B 0,C 180,E1 -18276.216,E2 -18276.216} C_VEL
LIN {X 0,Y 270.025,Z 377.572,A -85,B 0,C 180,E1 -18277.479,E2 -18277.479} C_VEL
LIN {X 0,Y 270.995,Z 365.921,A -85,B 0,C 180,E1 -18278.578,E2 -18278.578} C_VEL
LIN {X 0,Y 271.959,Z 353.108,A -85,B 0,C 180,E1 -18279.437,E2 -18279.437} C_VEL
LIN {X 0,Y 272.58,Z 339.684,A -85,B 0,C 180,E1 -18280.024,E2 -18280.024} C_VEL
LIN {X 0,Y 274.646,Z 264.358,A -85,B 0,C 180,E1 -18281.965,E2 -18281.965} C_VEL
LIN {X 0,Y 266.121,Z 243.605,A -85,B 0,C 180,E1 -18283.28,E2 -18283.28} C_VEL
LIN {X 0,Y 263.469,Z 237.413,A -85,B 0,C 180,E1 -18283.702,E2 -18283.702} C_VEL
LIN {X 0,Y 263.314,Z 236.685,A -85,B 0,C 180,E1 -18283.775,E2 -18283.775} C_VEL
LIN {X 0,Y 263.276,Z 236.689,A -85,B 0,C 180,E1 -18287.078,E2 -18287.078} C_VEL
LIN {X 0,Y 263.218,Z 236.697,A -85,B 0,C 180,E1 -18290.849,E2 -18290.849} C_VEL
LIN {X 0,Y 263.13,Z 236.707,A -85,B 0,C 180,E1 -18295.301,E2 -18295.301} C_VEL
LIN {X 0,Y 263.124,Z 236.708,A -85,B 0,C 180,E1 -18298.738,E2 -18298.738} C_VEL
LIN {X 0,Y 263.132,Z 236.708,A -85,B 0,C 180,E1 -18302.29,E2 -18302.29} C_VEL
LIN {X 0,Y 263.18,Z 236.696,A -85,B 0,C 180,E1 -18306.761,E2 -18306.761} C_VEL
LIN {X 0,Y 263.097,Z 236.712,A -85,B 0,C 180,E1 -18309.876,E2 -18309.876} C_VEL
LIN {X 0,Y 263.083,Z 236.71,A -85,B 0,C 180,E1 -18313.995,E2 -18313.995} C_VEL
LIN {X 0,Y 263.081,Z 236.711,A -85,B 0,C 180,E1 -18318.097,E2 -18318.097} C_VEL
LIN {X 0,Y 263.11,Z 236.699,A -85,B 0,C 180,E1 -18322.094,E2 -18322.094} C_VEL
LIN {X 0,Y 263.158,Z 236.702,A -85,B 0,C 180,E1 -18325.886,E2 -18325.886} C_VEL
LIN {X 0,Y 263.116,Z 236.702,A -85,B 0,C 180,E1 -18329.502,E2 -18329.502} C_VEL
LIN {X 0,Y 263.199,Z 236.688,A -85,B 0,C 180,E1 -18333.859,E2 -18333.859} C_VEL
LIN {X 0,Y 263.256,Z 236.822,A -85,B 0,C 180,E1 -18334.402,E2 -18334.402} C_VEL
LIN {X 0,Y 270.336,Z 263.945,A -85,B 0,C 180,E1 -18335.859,E2 -18335.859} C_VEL
LIN {X 0,Y 267.931,Z 324.926,A -85,B 0,C 180,E1 -18338.393,E2 -18338.393} C_VEL
LIN {X 0,Y 267.038,Z 330.675,A -85,B 0,C 180,E1 -18338.617,E2 -18338.617} C_VEL
LIN {X 0,Y 261.143,Z 347.23,A -85,B 0,C 180,E1 -18339.303,E2 -18339.303} C_VEL
LIN {X 0,Y 259.848,Z 352.789,A -85,B 0,C 180,E1 -18339.639,E2 -18339.639} C_VEL
LIN {X 0,Y 259.667,Z 354.656,A -85,B 0,C 180,E1 -18339.772,E2 -18339.772} C_VEL
LIN {X 0,Y 258.864,Z 368.996,A -85,B 0,C 180,E1 -18340.986,E2 -18340.986} C_VEL
LIN {X 0,Y 257.897,Z 382.495,A -85,B 0,C 180,E1 -18342.519,E2 -18342.519} C_VEL
LIN {X 0,Y 256.993,Z 393.769,A -85,B 0,C 180,E1 -18344.129,E2 -18344.129} C_VEL
LIN {X 0,Y 256.219,Z 404.932,A -85,B 0,C 180,E1 -18346.112,E2 -18346.112} C_VEL
LIN {X 0,Y 255.432,Z 414.062,A -85,B 0,C 180,E1 -18348.091,E2 -18348.091} C_VEL
LIN {X 0,Y 254.868,Z 422.976,A -85,B 0,C 180,E1 -18350.476,E2 -18350.476} C_VEL
LIN {X 0,Y 254.45,Z 430.158,A -85,B 0,C 180,E1 -18352.86,E2 -18352.86} C_VEL
LIN {X 0,Y 254.19,Z 435.913,A -85,B 0,C 180,E1 -18355.242,E2 -18355.242} C_VEL
LIN {X 0,Y 254.199,Z 440.404,A -85,B 0,C 180,E1 -18357.623,E2 -18357.623} C_VEL
LIN {X 0,Y 254.191,Z 443.769,A -85,B 0,C 180,E1 -18360,E2 -18360} C_VEL
LIN {X 0,Y 254.355,Z 445.443,A -85,B 0,C 180,E1 -18361.583,E2 -18361.583} C_VEL
LIN {X 0,Y 255.09,Z 447.516,A -85,B 0,C 180,E1 -18364.741,E2 -18364.741} C_VEL
LIN {X 0,Y 255.628,Z 447.955,A -85,B 0,C 180,E1 -18366.313,E2 -18366.313} C_VEL
LIN {X 0,Y 256.117,Z 447.97,A -85,B 0,C 180,E1 -18367.886,E2 -18367.886} C_VEL
LIN {X 0,Y 256.795,Z 447.58,A -85,B 0,C 180,E1 -18369.451,E2 -18369.451} C_VEL
LIN {X 0,Y 258.005,Z 446.766,A -85,B 0,C 180,E1 -18370.992,E2 -18370.992} C_VEL
LIN {X 0,Y 259.533,Z 445.233,A -85,B 0,C 180,E1 -18372.869,E2 -18372.869} C_VEL
LIN {X 0,Y 262.177,Z 441.863,A -85,B 0,C 180,E1 -18375.549,E2 -18375.549} C_VEL
LIN {X 0,Y 264.815,Z 437.94,A -85,B 0,C 180,E1 -18377.77,E2 -18377.77} C_VEL
LIN {X 0,Y 267.904,Z 432.906,A -85,B 0,C 180,E1 -18379.94,E2 -18379.94} C_VEL
LIN {X 0,Y 271.987,Z 425.514,A -85,B 0,C 180,E1 -18382.404,E2 -18382.404} C_VEL
LIN {X 0,Y 275.931,Z 417.555,A -85,B 0,C 180,E1 -18384.449,E2 -18384.449} C_VEL
LIN {X 0,Y 280.312,Z 407.838,A -85,B 0,C 180,E1 -18386.425,E2 -18386.425} C_VEL
LIN {X 0,Y 284.615,Z 396.917,A -85,B 0,C 180,E1 -18388.18,E2 -18388.18} C_VEL
LIN {X 0,Y 288.372,Z 386.077,A -85,B 0,C 180,E1 -18389.572,E2 -18389.572} C_VEL
LIN {X 0,Y 292.338,Z 372.548,A -85,B 0,C 180,E1 -18390.922,E2 -18390.922} C_VEL
LIN {X 0,Y 295.349,Z 360.091,A -85,B 0,C 180,E1 -18391.868,E2 -18391.868} C_VEL
LIN {X 0,Y 298.25,Z 344.739,A -85,B 0,C 180,E1 -18392.718,E2 -18392.718} C_VEL
LIN {X 0,Y 304.798,Z 306.821,A -85,B 0,C 180,E1 -18394.364,E2 -18394.364} C_VEL
LIN {X 0,Y 302.677,Z 302.512,A -85,B 0,C 180,E1 -18396.007,E2 -18396.007} C_VEL
LIN {X 0,Y 301.41,Z 300.144,A -85,B 0,C 180,E1 -18397.155,E2 -18397.155} C_VEL
LIN {X 0,Y 299.886,Z 297.467,A -85,B 0,C 180,E1 -18398.863,E2 -18398.863} C_VEL
LIN {X 0,Y 298.214,Z 295.285,A -85,B 0,C 180,E1 -18401.672,E2 -18401.672} C_VEL
LIN {X 0,Y 297.627,Z 295.333,A -85,B 0,C 180,E1 -18404.146,E2 -18404.146} C_VEL
LIN {X 0,Y 297.99,Z 296.732,A -85,B 0,C 180,E1 -18406.563,E2 -18406.563} C_VEL
LIN {X 0,Y 299.437,Z 301.463,A -85,B 0,C 180,E1 -18409.602,E2 -18409.602} C_VEL
LIN {X 0,Y 300.165,Z 303.442,A -85,B 0,C 180,E1 -18410.542,E2 -18410.542} C_VEL
LIN {X 0,Y 301.674,Z 308.117,A -85,B 0,C 180,E1 -18412.226,E2 -18412.226} C_VEL
LIN {X 0,Y 303.108,Z 312.845,A -85,B 0,C 180,E1 -18413.569,E2 -18413.569} C_VEL
LIN {X 0,Y 303.313,Z 314.221,A -85,B 0,C 180,E1 -18413.834,E2 -18413.834} C_VEL
LIN {X 0,Y 303.153,Z 319.853,A -85,B 0,C 180,E1 -18414.427,E2 -18414.427} C_VEL
LIN {X 0,Y 295.417,Z 365.483,A -85,B 0,C 180,E1 -18416.468,E2 -18416.468} C_VEL
LIN {X 0,Y 292.343,Z 378.71,A -85,B 0,C 180,E1 -18417.252,E2 -18417.252} C_VEL
LIN {X 0,Y 288.092,Z 393.163,A -85,B 0,C 180,E1 -18418.364,E2 -18418.364} C_VEL
LIN {X 0,Y 283.362,Z 407.091,A -85,B 0,C 180,E1 -18419.85,E2 -18419.85} C_VEL
LIN {X 0,Y 278.933,Z 418.385,A -85,B 0,C 180,E1 -18421.396,E2 -18421.396} C_VEL
LIN {X 0,Y 274.987,Z 427.796,A -85,B 0,C 180,E1 -18423.02,E2 -18423.02} C_VEL
LIN {X 0,Y 270.695,Z 437.259,A -85,B 0,C 180,E1 -18425.044,E2 -18425.044} C_VEL
LIN {X 0,Y 266.492,Z 445.798,A -85,B 0,C 180,E1 -18427.373,E2 -18427.373} C_VEL
LIN {X 0,Y 262.992,Z 452.452,A -85,B 0,C 180,E1 -18429.67,E2 -18429.67} C_VEL
LIN {X 0,Y 260.443,Z 457.505,A -85,B 0,C 180,E1 -18431.919,E2 -18431.919} C_VEL
LIN {X 0,Y 258.157,Z 461.541,A -85,B 0,C 180,E1 -18434.201,E2 -18434.201} C_VEL
LIN {X 0,Y 256.898,Z 463.7,A -85,B 0,C 180,E1 -18435.745,E2 -18435.745} C_VEL
LIN {X 0,Y 255.97,Z 465.434,A -85,B 0,C 180,E1 -18437.31,E2 -18437.31} C_VEL
LIN {X 0,Y 254.672,Z 467.65,A -85,B 0,C 180,E1 -18440.467,E2 -18440.467} C_VEL
LIN {X 0,Y 254.124,Z 468.313,A -85,B 0,C 180,E1 -18443.647,E2 -18443.647} C_VEL
LIN {X 0,Y 254.09,Z 468.03,A -85,B 0,C 180,E1 -18445.238,E2 -18445.238} C_VEL
LIN {X 0,Y 254.245,Z 466.519,A -85,B 0,C 180,E1 -18448.018,E2 -18448.018} C_VEL
